   1:  PR[GP1:91,2] = PR[GP1:90,2] + -31.006;
   1:L PR[91] 10mm/sec CNT100;
   1:  PR[GP1:91,1] = PR[GP1:90,1] + -0.266;
   1:  PR[GP1:91,2] = PR[GP1:90,2] + -30.252;
   1:L PR[91] 10mm/sec CNT100;
   1:  PR[GP1:91,1] = PR[GP1:90,1] + 0.371;
   1:  PR[GP1:91,2] = PR[GP1:90,2] + -31.082;
   1:  PR[GP1:91,3] = PR[GP1:90,3] + 67.405;
   1:L PR[91] 10mm/sec CNT100;
   1:  PR[GP1:91,1] = PR[GP1:90,1] + 7.171;
   1:  PR[GP1:91,2] = PR[GP1:90,2] + -35.054;
   1:L PR[91] 10mm/sec CNT100;
   1:  PR[GP1:91,1] = PR[GP1:90,1] + 10.495;
   1:  PR[GP1:91,2] = PR[GP1:90,2] + -36.009;
   1:L PR[91] 10mm/sec CNT100;
   1:  PR[GP1:91,1] = PR[GP1:90,1] + 18.333;
   1:  PR[GP1:91,2] = PR[GP1:90,2] + -37.802;
   1:L PR[91] 10mm/sec CNT100;
   1:  PR[GP1:91,1] = PR[GP1:90,1] + 22.053;
   1:  PR[GP1:91,2] = PR[GP1:90,2] + -38.049;
   1:L PR[91] 10mm/sec CNT100;
   1:  PR[GP1:91,1] = PR[GP1:90,1] + 26.238;
   1:  PR[GP1:91,2] = PR[GP1:90,2] + -37.472;
   1:L PR[91] 10mm/sec CNT100;
   1:  PR[GP1:91,1] = PR[GP1:90,1] + 33.369;
   1:  PR[GP1:91,2] = PR[GP1:90,2] + -36.778;
   1:L PR[91] 10mm/sec CNT100;
   1:  PR[GP1:91,1] = PR[GP1:90,1] + 37.578;
   1:  PR[GP1:91,2] = PR[GP1:90,2] + -35.242;
   1:L PR[91] 10mm/sec CNT100;
   1:  PR[GP1:91,1] = PR[GP1:90,1] + 43.414;
   1:  PR[GP1:91,2] = PR[GP1:90,2] + -32.676;
   1:L PR[91] 10mm/sec CNT100;
   1:  PR[GP1:91,1] = PR[GP1:90,1] + 47.360;
   1:  PR[GP1:91,2] = PR[GP1:90,2] + -30.200;
   1:L PR[91] 10mm/sec CNT100;
   1:  PR[GP1:91,1] = PR[GP1:90,1] + 50.959;
   1:  PR[GP1:91,2] = PR[GP1:90,2] + -26.692;
   1:L PR[91] 10mm/sec CNT100;
   1:  PR[GP1:91,1] = PR[GP1:90,1] + 54.991;
   1:  PR[GP1:91,2] = PR[GP1:90,2] + -23.025;
   1:L PR[91] 10mm/sec CNT100;
   1:  PR[GP1:91,1] = PR[GP1:90,1] + 57.831;
   1:  PR[GP1:91,2] = PR[GP1:90,2] + -18.619;
   1:L PR[91] 10mm/sec CNT100;
   1:  PR[GP1:91,1] = PR[GP1:90,1] + 60.207;
   1:  PR[GP1:91,2] = PR[GP1:90,2] + -14.324;
   1:L PR[91] 10mm/sec CNT100;
   1:  PR[GP1:91,1] = PR[GP1:90,1] + 61.985;
   1:  PR[GP1:91,2] = PR[GP1:90,2] + -9.491;
   1:L PR[91] 10mm/sec CNT100;
   1:  PR[GP1:91,1] = PR[GP1:90,1] + 62.584;
   1:  PR[GP1:91,2] = PR[GP1:90,2] + -4.219;
   1:L PR[91] 10mm/sec CNT100;
   1:  PR[GP1:91,1] = PR[GP1:90,1] + 63.354;
   1:  PR[GP1:91,2] = PR[GP1:90,2] + 0.296;
   1:L PR[91] 10mm/sec CNT100;
   1:  PR[GP1:91,1] = PR[GP1:90,1] + 62.767;
   1:  PR[GP1:91,2] = PR[GP1:90,2] + 5.490;
   1:L PR[91] 10mm/sec CNT100;
   1:  PR[GP1:91,1] = PR[GP1:90,1] + 61.988;
   1:  PR[GP1:91,2] = PR[GP1:90,2] + 10.042;
   1:L PR[91] 10mm/sec CNT100;
   1:  PR[GP1:91,1] = PR[GP1:90,1] + 60.204;
   1:  PR[GP1:91,2] = PR[GP1:90,2] + 14.892;
   1:L PR[91] 10mm/sec CNT100;
   1:  PR[GP1:91,1] = PR[GP1:90,1] + 57.818;
   1:  PR[GP1:91,2] = PR[GP1:90,2] + 19.195;
   1:L PR[91] 10mm/sec CNT100;
   1:  PR[GP1:91,1] = PR[GP1:90,1] + 54.971;
   1:  PR[GP1:91,2] = PR[GP1:90,2] + 23.610;
   1:L PR[91] 10mm/sec CNT100;
   1:  PR[GP1:91,1] = PR[GP1:90,1] + 51.546;
   1:  PR[GP1:91,2] = PR[GP1:90,2] + 26.964;
   1:L PR[91] 10mm/sec CNT100;
   1:  PR[GP1:91,1] = PR[GP1:90,1] + 47.338;
   1:  PR[GP1:91,2] = PR[GP1:90,2] + 30.773;
   1:L PR[91] 10mm/sec CNT100;
   1:  PR[GP1:91,1] = PR[GP1:90,1] + 43.381;
   1:  PR[GP1:91,2] = PR[GP1:90,2] + 33.255;
   1:L PR[91] 10mm/sec CNT100;
   1:  PR[GP1:91,1] = PR[GP1:90,1] + 37.523;
   1:  PR[GP1:91,2] = PR[GP1:90,2] + 35.815;
   1:L PR[91] 10mm/sec CNT100;
   1:  PR[GP1:91,1] = PR[GP1:90,1] + 33.299;
   1:  PR[GP1:91,2] = PR[GP1:90,2] + 37.356;
   1:L PR[91] 10mm/sec CNT100;
   1:  PR[GP1:91,1] = PR[GP1:90,1] + 29.302;
   1:  PR[GP1:91,2] = PR[GP1:90,2] + 37.923;
   1:L PR[91] 10mm/sec CNT100;
   1:  PR[GP1:91,1] = PR[GP1:90,1] + 21.984;
   1:  PR[GP1:91,2] = PR[GP1:90,2] + 38.603;
   1:L PR[91] 10mm/sec CNT100;
   1:  PR[GP1:91,1] = PR[GP1:90,1] + 18.251;
   1:  PR[GP1:91,2] = PR[GP1:90,2] + 38.355;
   1:L PR[91] 10mm/sec CNT100;
   1:  PR[GP1:91,1] = PR[GP1:90,1] + 10.284;
   1:  PR[GP1:91,2] = PR[GP1:90,2] + 36.473;
   1:L PR[91] 10mm/sec CNT100;
   1:  PR[GP1:91,1] = PR[GP1:90,1] + 7.009;
   1:  PR[GP1:91,2] = PR[GP1:90,2] + 35.532;
   1:L PR[91] 10mm/sec CNT100;
   1:  PR[GP1:91,1] = PR[GP1:90,1] + 5.914;
   1:  PR[GP1:91,2] = PR[GP1:90,2] + 34.958;
   1:L PR[91] 10mm/sec CNT100;
   1:  PR[GP1:91,1] = PR[GP1:90,1] + 3.650;
   1:  PR[GP1:91,2] = PR[GP1:90,2] + 33.735;
   1:L PR[91] 10mm/sec CNT100;
   1:  PR[GP1:91,1] = PR[GP1:90,1] + -0.263;
   1:  PR[GP1:91,2] = PR[GP1:90,2] + 30.552;
   1:L PR[91] 10mm/sec CNT100;
   1:  PR[GP1:91,1] = PR[GP1:90,1] + -4.166;
   1:  PR[GP1:91,2] = PR[GP1:90,2] + 33.726;
   1:L PR[91] 10mm/sec CNT100;
   1:  PR[GP1:91,1] = PR[GP1:90,1] + -6.444;
   1:  PR[GP1:91,2] = PR[GP1:90,2] + 34.959;
   1:L PR[91] 10mm/sec CNT100;
   1:  PR[GP1:91,1] = PR[GP1:90,1] + -7.536;
   1:  PR[GP1:91,2] = PR[GP1:90,2] + 35.533;
   1:L PR[91] 10mm/sec CNT100;
   1:  PR[GP1:91,1] = PR[GP1:90,1] + -10.806;
   1:  PR[GP1:91,2] = PR[GP1:90,2] + 36.474;
   1:L PR[91] 10mm/sec CNT100;
   1:  PR[GP1:91,1] = PR[GP1:90,1] + -18.776;
   1:  PR[GP1:91,2] = PR[GP1:90,2] + 38.355;
   1:L PR[91] 10mm/sec CNT100;
   1:  PR[GP1:91,1] = PR[GP1:90,1] + -22.506;
   1:  PR[GP1:91,2] = PR[GP1:90,2] + 38.601;
   1:L PR[91] 10mm/sec CNT100;
   1:  PR[GP1:91,1] = PR[GP1:90,1] + -26.707;
   1:  PR[GP1:91,2] = PR[GP1:90,2] + 38.020;
   1:L PR[91] 10mm/sec CNT100;
   1:  PR[GP1:91,1] = PR[GP1:90,1] + -33.861;
   1:  PR[GP1:91,2] = PR[GP1:90,2] + 37.347;
   1:L PR[91] 10mm/sec CNT100;
   1:  PR[GP1:91,1] = PR[GP1:90,1] + -38.066;
   1:  PR[GP1:91,2] = PR[GP1:90,2] + 35.807;
   1:L PR[91] 10mm/sec CNT100;
   1:  PR[GP1:91,1] = PR[GP1:90,1] + -43.923;
   1:  PR[GP1:91,2] = PR[GP1:90,2] + 33.246;
   1:L PR[91] 10mm/sec CNT100;
   1:  PR[GP1:91,1] = PR[GP1:90,1] + -47.894;
   1:  PR[GP1:91,2] = PR[GP1:90,2] + 30.742;
   1:L PR[91] 10mm/sec CNT100;
   1:  PR[GP1:91,1] = PR[GP1:90,1] + -51.502;
   1:  PR[GP1:91,2] = PR[GP1:90,2] + 27.221;
   1:L PR[91] 10mm/sec CNT100;
   1:  PR[GP1:91,1] = PR[GP1:90,1] + -55.548;
   1:  PR[GP1:91,2] = PR[GP1:90,2] + 23.557;
   1:L PR[91] 10mm/sec CNT100;
   1:  PR[GP1:91,1] = PR[GP1:90,1] + -58.358;
   1:  PR[GP1:91,2] = PR[GP1:90,2] + 19.171;
   1:L PR[91] 10mm/sec CNT100;
   1:  PR[GP1:91,1] = PR[GP1:90,1] + -60.744;
   1:  PR[GP1:91,2] = PR[GP1:90,2] + 14.862;
   1:L PR[91] 10mm/sec CNT100;
   1:  PR[GP1:91,1] = PR[GP1:90,1] + -62.529;
   1:  PR[GP1:91,2] = PR[GP1:90,2] + 9.943;
   1:L PR[91] 10mm/sec CNT100;
   1:  PR[GP1:91,1] = PR[GP1:90,1] + -63.107;
   1:  PR[GP1:91,2] = PR[GP1:90,2] + 4.782;
   1:L PR[91] 10mm/sec CNT100;
   1:  PR[GP1:91,1] = PR[GP1:90,1] + -63.881;
   1:  PR[GP1:91,2] = PR[GP1:90,2] + 0.261;
   1:L PR[91] 10mm/sec CNT100;
   1:  PR[GP1:91,1] = PR[GP1:90,1] + -63.314;
   1:  PR[GP1:91,2] = PR[GP1:90,2] + -4.822;
   1:L PR[91] 10mm/sec CNT100;
   1:  PR[GP1:91,1] = PR[GP1:90,1] + -62.538;
   1:  PR[GP1:91,2] = PR[GP1:90,2] + -9.359;
   1:L PR[91] 10mm/sec CNT100;
   1:  PR[GP1:91,1] = PR[GP1:90,1] + -60.747;
   1:  PR[GP1:91,2] = PR[GP1:90,2] + -14.294;
   1:L PR[91] 10mm/sec CNT100;
   1:  PR[GP1:91,1] = PR[GP1:90,1] + -58.372;
   1:  PR[GP1:91,2] = PR[GP1:90,2] + -18.596;
   1:L PR[91] 10mm/sec CNT100;
   1:  PR[GP1:91,1] = PR[GP1:90,1] + -55.555;
   1:  PR[GP1:91,2] = PR[GP1:90,2] + -22.992;
   1:L PR[91] 10mm/sec CNT100;
   1:  PR[GP1:91,1] = PR[GP1:90,1] + -52.126;
   1:  PR[GP1:91,2] = PR[GP1:90,2] + -26.357;
   1:L PR[91] 10mm/sec CNT100;
   1:  PR[GP1:91,1] = PR[GP1:90,1] + -47.936;
   1:  PR[GP1:91,2] = PR[GP1:90,2] + -30.157;
   1:L PR[91] 10mm/sec CNT100;
   1:  PR[GP1:91,1] = PR[GP1:90,1] + -43.956;
   1:  PR[GP1:91,2] = PR[GP1:90,2] + -32.667;
   1:L PR[91] 10mm/sec CNT100;
   1:  PR[GP1:91,1] = PR[GP1:90,1] + -38.121;
   1:  PR[GP1:91,2] = PR[GP1:90,2] + -35.235;
   1:L PR[91] 10mm/sec CNT100;
   1:  PR[GP1:91,1] = PR[GP1:90,1] + -33.905;
   1:  PR[GP1:91,2] = PR[GP1:90,2] + -36.779;
   1:L PR[91] 10mm/sec CNT100;
   1:  PR[GP1:91,1] = PR[GP1:90,1] + -29.897;
   1:  PR[GP1:91,2] = PR[GP1:90,2] + -37.349;
   1:L PR[91] 10mm/sec CNT100;
   1:  PR[GP1:91,1] = PR[GP1:90,1] + -22.602;
   1:  PR[GP1:91,2] = PR[GP1:90,2] + -38.049;
   1:L PR[91] 10mm/sec CNT100;
   1:  PR[GP1:91,1] = PR[GP1:90,1] + -18.858;
   1:  PR[GP1:91,2] = PR[GP1:90,2] + -37.802;
   1:L PR[91] 10mm/sec CNT100;
   1:  PR[GP1:91,1] = PR[GP1:90,1] + -11.020;
   1:  PR[GP1:91,2] = PR[GP1:90,2] + -36.009;
   1:L PR[91] 10mm/sec CNT100;
   1:  PR[GP1:91,1] = PR[GP1:90,1] + -7.700;
   1:  PR[GP1:91,2] = PR[GP1:90,2] + -35.055;
   1:L PR[91] 10mm/sec CNT100;
   1:  PR[GP1:91,1] = PR[GP1:90,1] + -0.903;
   1:  PR[GP1:91,2] = PR[GP1:90,2] + -31.081;
   1:L PR[91] 10mm/sec CNT100;
   1:  PR[GP1:91,1] = PR[GP1:90,1] + -0.266;
   1:  PR[GP1:91,2] = PR[GP1:90,2] + -30.532;
   1:L PR[91] 10mm/sec CNT100;
   1:  PR[GP1:91,1] = PR[GP1:90,1] + 0.126;
   1:  PR[GP1:91,2] = PR[GP1:90,2] + -31.151;
   1:  PR[GP1:91,3] = PR[GP1:90,3] + 68.015;
   1:L PR[91] 10mm/sec CNT100;
   1:  PR[GP1:91,1] = PR[GP1:90,1] + 6.916;
   1:  PR[GP1:91,2] = PR[GP1:90,2] + -35.123;
   1:L PR[91] 10mm/sec CNT100;
   1:  PR[GP1:91,1] = PR[GP1:90,1] + 10.120;
   1:  PR[GP1:91,2] = PR[GP1:90,2] + -36.043;
   1:L PR[91] 10mm/sec CNT100;
   1:  PR[GP1:91,1] = PR[GP1:90,1] + 18.156;
   1:  PR[GP1:91,2] = PR[GP1:90,2] + -37.882;
   1:L PR[91] 10mm/sec CNT100;
   1:  PR[GP1:91,1] = PR[GP1:90,1] + 21.753;
   1:  PR[GP1:91,2] = PR[GP1:90,2] + -38.121;
   1:L PR[91] 10mm/sec CNT100;
   1:  PR[GP1:91,1] = PR[GP1:90,1] + 25.802;
   1:  PR[GP1:91,2] = PR[GP1:90,2] + -37.562;
   1:L PR[91] 10mm/sec CNT100;
   1:  PR[GP1:91,1] = PR[GP1:90,1] + 33.152;
   1:  PR[GP1:91,2] = PR[GP1:90,2] + -36.848;
   1:L PR[91] 10mm/sec CNT100;
   1:  PR[GP1:91,1] = PR[GP1:90,1] + 37.234;
   1:  PR[GP1:91,2] = PR[GP1:90,2] + -35.358;
   1:L PR[91] 10mm/sec CNT100;
   1:  PR[GP1:91,1] = PR[GP1:90,1] + 43.269;
   1:  PR[GP1:91,2] = PR[GP1:90,2] + -32.704;
   1:L PR[91] 10mm/sec CNT100;
   1:  PR[GP1:91,1] = PR[GP1:90,1] + 47.105;
   1:  PR[GP1:91,2] = PR[GP1:90,2] + -30.297;
   1:L PR[91] 10mm/sec CNT100;
   1:  PR[GP1:91,1] = PR[GP1:90,1] + 50.604;
   1:  PR[GP1:91,2] = PR[GP1:90,2] + -26.887;
   1:L PR[91] 10mm/sec CNT100;
   1:  PR[GP1:91,1] = PR[GP1:90,1] + 54.804;
   1:  PR[GP1:91,2] = PR[GP1:90,2] + -23.066;
   1:L PR[91] 10mm/sec CNT100;
   1:  PR[GP1:91,1] = PR[GP1:90,1] + 57.569;
   1:  PR[GP1:91,2] = PR[GP1:90,2] + -18.777;
   1:L PR[91] 10mm/sec CNT100;
   1:  PR[GP1:91,1] = PR[GP1:90,1] + 60.053;
   1:  PR[GP1:91,2] = PR[GP1:90,2] + -14.287;
   1:L PR[91] 10mm/sec CNT100;
   1:  PR[GP1:91,1] = PR[GP1:90,1] + 61.786;
   1:  PR[GP1:91,2] = PR[GP1:90,2] + -9.578;
   1:L PR[91] 10mm/sec CNT100;
   1:  PR[GP1:91,1] = PR[GP1:90,1] + 62.370;
   1:  PR[GP1:91,2] = PR[GP1:90,2] + -4.439;
   1:L PR[91] 10mm/sec CNT100;
   1:  PR[GP1:91,1] = PR[GP1:90,1] + 63.177;
   1:  PR[GP1:91,2] = PR[GP1:90,2] + 0.296;
   1:L PR[91] 10mm/sec CNT100;
   1:  PR[GP1:91,1] = PR[GP1:90,1] + 62.605;
   1:  PR[GP1:91,2] = PR[GP1:90,2] + 5.360;
   1:L PR[91] 10mm/sec CNT100;
   1:  PR[GP1:91,1] = PR[GP1:90,1] + 61.788;
   1:  PR[GP1:91,2] = PR[GP1:90,2] + 10.130;
   1:L PR[91] 10mm/sec CNT100;
   1:  PR[GP1:91,1] = PR[GP1:90,1] + 60.050;
   1:  PR[GP1:91,2] = PR[GP1:90,2] + 14.855;
   1:L PR[91] 10mm/sec CNT100;
   1:  PR[GP1:91,1] = PR[GP1:90,1] + 57.555;
   1:  PR[GP1:91,2] = PR[GP1:90,2] + 19.353;
   1:L PR[91] 10mm/sec CNT100;
   1:  PR[GP1:91,1] = PR[GP1:90,1] + 54.783;
   1:  PR[GP1:91,2] = PR[GP1:90,2] + 23.653;
   1:L PR[91] 10mm/sec CNT100;
   1:  PR[GP1:91,1] = PR[GP1:90,1] + 51.448;
   1:  PR[GP1:91,2] = PR[GP1:90,2] + 26.918;
   1:L PR[91] 10mm/sec CNT100;
   1:  PR[GP1:91,1] = PR[GP1:90,1] + 47.081;
   1:  PR[GP1:91,2] = PR[GP1:90,2] + 30.871;
   1:L PR[91] 10mm/sec CNT100;
   1:  PR[GP1:91,1] = PR[GP1:90,1] + 43.235;
   1:  PR[GP1:91,2] = PR[GP1:90,2] + 33.284;
   1:L PR[91] 10mm/sec CNT100;
   1:  PR[GP1:91,1] = PR[GP1:90,1] + 37.177;
   1:  PR[GP1:91,2] = PR[GP1:90,2] + 35.931;
   1:L PR[91] 10mm/sec CNT100;
   1:  PR[GP1:91,1] = PR[GP1:90,1] + 33.080;
   1:  PR[GP1:91,2] = PR[GP1:90,2] + 37.426;
   1:L PR[91] 10mm/sec CNT100;
   1:  PR[GP1:91,1] = PR[GP1:90,1] + 29.203;
   1:  PR[GP1:91,2] = PR[GP1:90,2] + 37.976;
   1:L PR[91] 10mm/sec CNT100;
   1:  PR[GP1:91,1] = PR[GP1:90,1] + 21.682;
   1:  PR[GP1:91,2] = PR[GP1:90,2] + 38.675;
   1:L PR[91] 10mm/sec CNT100;
   1:  PR[GP1:91,1] = PR[GP1:90,1] + 18.072;
   1:  PR[GP1:91,2] = PR[GP1:90,2] + 38.435;
   1:L PR[91] 10mm/sec CNT100;
   1:  PR[GP1:91,1] = PR[GP1:90,1] + 9.904;
   1:  PR[GP1:91,2] = PR[GP1:90,2] + 36.506;
   1:L PR[91] 10mm/sec CNT100;
   1:  PR[GP1:91,1] = PR[GP1:90,1] + 6.751;
   1:  PR[GP1:91,2] = PR[GP1:90,2] + 35.599;
   1:L PR[91] 10mm/sec CNT100;
   1:  PR[GP1:91,1] = PR[GP1:90,1] + 5.630;
   1:  PR[GP1:91,2] = PR[GP1:90,2] + 35.011;
   1:L PR[91] 10mm/sec CNT100;
   1:  PR[GP1:91,1] = PR[GP1:90,1] + 3.477;
   1:  PR[GP1:91,2] = PR[GP1:90,2] + 33.849;
   1:L PR[91] 10mm/sec CNT100;
   1:  PR[GP1:91,1] = PR[GP1:90,1] + -0.263;
   1:  PR[GP1:91,2] = PR[GP1:90,2] + 30.807;
   1:L PR[91] 10mm/sec CNT100;
   1:  PR[GP1:91,1] = PR[GP1:90,1] + -3.994;
   1:  PR[GP1:91,2] = PR[GP1:90,2] + 33.840;
   1:L PR[91] 10mm/sec CNT100;
   1:  PR[GP1:91,1] = PR[GP1:90,1] + -6.158;
   1:  PR[GP1:91,2] = PR[GP1:90,2] + 35.012;
   1:L PR[91] 10mm/sec CNT100;
   1:  PR[GP1:91,1] = PR[GP1:90,1] + -7.277;
   1:  PR[GP1:91,2] = PR[GP1:90,2] + 35.601;
   1:L PR[91] 10mm/sec CNT100;
   1:  PR[GP1:91,1] = PR[GP1:90,1] + -10.426;
   1:  PR[GP1:91,2] = PR[GP1:90,2] + 36.506;
   1:L PR[91] 10mm/sec CNT100;
   1:  PR[GP1:91,1] = PR[GP1:90,1] + -18.597;
   1:  PR[GP1:91,2] = PR[GP1:90,2] + 38.435;
   1:L PR[91] 10mm/sec CNT100;
   1:  PR[GP1:91,1] = PR[GP1:90,1] + -22.204;
   1:  PR[GP1:91,2] = PR[GP1:90,2] + 38.673;
   1:L PR[91] 10mm/sec CNT100;
   1:  PR[GP1:91,1] = PR[GP1:90,1] + -26.268;
   1:  PR[GP1:91,2] = PR[GP1:90,2] + 38.111;
   1:L PR[91] 10mm/sec CNT100;
   1:  PR[GP1:91,1] = PR[GP1:90,1] + -33.641;
   1:  PR[GP1:91,2] = PR[GP1:90,2] + 37.417;
   1:L PR[91] 10mm/sec CNT100;
   1:  PR[GP1:91,1] = PR[GP1:90,1] + -37.719;
   1:  PR[GP1:91,2] = PR[GP1:90,2] + 35.924;
   1:L PR[91] 10mm/sec CNT100;
   1:  PR[GP1:91,1] = PR[GP1:90,1] + -43.777;
   1:  PR[GP1:91,2] = PR[GP1:90,2] + 33.275;
   1:L PR[91] 10mm/sec CNT100;
   1:  PR[GP1:91,1] = PR[GP1:90,1] + -47.636;
   1:  PR[GP1:91,2] = PR[GP1:90,2] + 30.842;
   1:L PR[91] 10mm/sec CNT100;
   1:  PR[GP1:91,1] = PR[GP1:90,1] + -51.144;
   1:  PR[GP1:91,2] = PR[GP1:90,2] + 27.417;
   1:L PR[91] 10mm/sec CNT100;
   1:  PR[GP1:91,1] = PR[GP1:90,1] + -55.359;
   1:  PR[GP1:91,2] = PR[GP1:90,2] + 23.601;
   1:L PR[91] 10mm/sec CNT100;
   1:  PR[GP1:91,1] = PR[GP1:90,1] + -58.095;
   1:  PR[GP1:91,2] = PR[GP1:90,2] + 19.331;
   1:L PR[91] 10mm/sec CNT100;
   1:  PR[GP1:91,1] = PR[GP1:90,1] + -60.589;
   1:  PR[GP1:91,2] = PR[GP1:90,2] + 14.826;
   1:L PR[91] 10mm/sec CNT100;
   1:  PR[GP1:91,1] = PR[GP1:90,1] + -62.329;
   1:  PR[GP1:91,2] = PR[GP1:90,2] + 10.033;
   1:L PR[91] 10mm/sec CNT100;
   1:  PR[GP1:91,1] = PR[GP1:90,1] + -62.892;
   1:  PR[GP1:91,2] = PR[GP1:90,2] + 5.002;
   1:L PR[91] 10mm/sec CNT100;
   1:  PR[GP1:91,1] = PR[GP1:90,1] + -63.704;
   1:  PR[GP1:91,2] = PR[GP1:90,2] + 0.261;
   1:L PR[91] 10mm/sec CNT100;
   1:  PR[GP1:91,1] = PR[GP1:90,1] + -63.151;
   1:  PR[GP1:91,2] = PR[GP1:90,2] + -4.694;
   1:L PR[91] 10mm/sec CNT100;
   1:  PR[GP1:91,1] = PR[GP1:90,1] + -62.338;
   1:  PR[GP1:91,2] = PR[GP1:90,2] + -9.448;
   1:L PR[91] 10mm/sec CNT100;
   1:  PR[GP1:91,1] = PR[GP1:90,1] + -60.593;
   1:  PR[GP1:91,2] = PR[GP1:90,2] + -14.258;
   1:L PR[91] 10mm/sec CNT100;
   1:  PR[GP1:91,1] = PR[GP1:90,1] + -58.109;
   1:  PR[GP1:91,2] = PR[GP1:90,2] + -18.754;
   1:L PR[91] 10mm/sec CNT100;
   1:  PR[GP1:91,1] = PR[GP1:90,1] + -55.367;
   1:  PR[GP1:91,2] = PR[GP1:90,2] + -23.035;
   1:L PR[91] 10mm/sec CNT100;
   1:  PR[GP1:91,1] = PR[GP1:90,1] + -52.028;
   1:  PR[GP1:91,2] = PR[GP1:90,2] + -26.311;
   1:L PR[91] 10mm/sec CNT100;
   1:  PR[GP1:91,1] = PR[GP1:90,1] + -47.680;
   1:  PR[GP1:91,2] = PR[GP1:90,2] + -30.256;
   1:L PR[91] 10mm/sec CNT100;
   1:  PR[GP1:91,1] = PR[GP1:90,1] + -43.811;
   1:  PR[GP1:91,2] = PR[GP1:90,2] + -32.695;
   1:L PR[91] 10mm/sec CNT100;
   1:  PR[GP1:91,1] = PR[GP1:90,1] + -37.777;
   1:  PR[GP1:91,2] = PR[GP1:90,2] + -35.351;
   1:L PR[91] 10mm/sec CNT100;
   1:  PR[GP1:91,1] = PR[GP1:90,1] + -33.687;
   1:  PR[GP1:91,2] = PR[GP1:90,2] + -36.849;
   1:L PR[91] 10mm/sec CNT100;
   1:  PR[GP1:91,1] = PR[GP1:90,1] + -29.799;
   1:  PR[GP1:91,2] = PR[GP1:90,2] + -37.402;
   1:L PR[91] 10mm/sec CNT100;
   1:  PR[GP1:91,1] = PR[GP1:90,1] + -22.302;
   1:  PR[GP1:91,2] = PR[GP1:90,2] + -38.121;
   1:L PR[91] 10mm/sec CNT100;
   1:  PR[GP1:91,1] = PR[GP1:90,1] + -18.681;
   1:  PR[GP1:91,2] = PR[GP1:90,2] + -37.882;
   1:L PR[91] 10mm/sec CNT100;
   1:  PR[GP1:91,1] = PR[GP1:90,1] + -10.645;
   1:  PR[GP1:91,2] = PR[GP1:90,2] + -36.044;
   1:L PR[91] 10mm/sec CNT100;
   1:  PR[GP1:91,1] = PR[GP1:90,1] + -7.446;
   1:  PR[GP1:91,2] = PR[GP1:90,2] + -35.125;
   1:L PR[91] 10mm/sec CNT100;
   1:  PR[GP1:91,1] = PR[GP1:90,1] + -0.659;
   1:  PR[GP1:91,2] = PR[GP1:90,2] + -31.150;
   1:L PR[91] 10mm/sec CNT100;
   1:  PR[GP1:91,1] = PR[GP1:90,1] + -0.266;
   1:  PR[GP1:91,2] = PR[GP1:90,2] + -30.811;
   1:L PR[91] 10mm/sec CNT100;
   1:  PR[GP1:91,1] = PR[GP1:90,1] + 6.662;
   1:  PR[GP1:91,2] = PR[GP1:90,2] + -35.193;
   1:  PR[GP1:91,3] = PR[GP1:90,3] + 68.625;
   1:L PR[91] 10mm/sec CNT100;
   1:  PR[GP1:91,1] = PR[GP1:90,1] + 9.744;
   1:  PR[GP1:91,2] = PR[GP1:90,2] + -36.078;
   1:L PR[91] 10mm/sec CNT100;
   1:  PR[GP1:91,1] = PR[GP1:90,1] + 17.979;
   1:  PR[GP1:91,2] = PR[GP1:90,2] + -37.962;
   1:L PR[91] 10mm/sec CNT100;
   1:  PR[GP1:91,1] = PR[GP1:90,1] + 21.453;
   1:  PR[GP1:91,2] = PR[GP1:90,2] + -38.193;
   1:L PR[91] 10mm/sec CNT100;
   1:  PR[GP1:91,1] = PR[GP1:90,1] + 25.366;
   1:  PR[GP1:91,2] = PR[GP1:90,2] + -37.653;
   1:L PR[91] 10mm/sec CNT100;
   1:  PR[GP1:91,1] = PR[GP1:90,1] + 32.934;
   1:  PR[GP1:91,2] = PR[GP1:90,2] + -36.918;
   1:L PR[91] 10mm/sec CNT100;
   1:  PR[GP1:91,1] = PR[GP1:90,1] + 36.890;
   1:  PR[GP1:91,2] = PR[GP1:90,2] + -35.474;
   1:L PR[91] 10mm/sec CNT100;
   1:  PR[GP1:91,1] = PR[GP1:90,1] + 43.124;
   1:  PR[GP1:91,2] = PR[GP1:90,2] + -32.732;
   1:L PR[91] 10mm/sec CNT100;
   1:  PR[GP1:91,1] = PR[GP1:90,1] + 46.849;
   1:  PR[GP1:91,2] = PR[GP1:90,2] + -30.395;
   1:L PR[91] 10mm/sec CNT100;
   1:  PR[GP1:91,1] = PR[GP1:90,1] + 50.249;
   1:  PR[GP1:91,2] = PR[GP1:90,2] + -27.081;
   1:L PR[91] 10mm/sec CNT100;
   1:  PR[GP1:91,1] = PR[GP1:90,1] + 54.617;
   1:  PR[GP1:91,2] = PR[GP1:90,2] + -23.108;
   1:L PR[91] 10mm/sec CNT100;
   1:  PR[GP1:91,1] = PR[GP1:90,1] + 57.308;
   1:  PR[GP1:91,2] = PR[GP1:90,2] + -18.935;
   1:L PR[91] 10mm/sec CNT100;
   1:  PR[GP1:91,1] = PR[GP1:90,1] + 59.899;
   1:  PR[GP1:91,2] = PR[GP1:90,2] + -14.251;
   1:L PR[91] 10mm/sec CNT100;
   1:  PR[GP1:91,1] = PR[GP1:90,1] + 61.586;
   1:  PR[GP1:91,2] = PR[GP1:90,2] + -9.664;
   1:L PR[91] 10mm/sec CNT100;
   1:  PR[GP1:91,1] = PR[GP1:90,1] + 62.155;
   1:  PR[GP1:91,2] = PR[GP1:90,2] + -4.659;
   1:L PR[91] 10mm/sec CNT100;
   1:  PR[GP1:91,1] = PR[GP1:90,1] + 63.000;
   1:  PR[GP1:91,2] = PR[GP1:90,2] + 0.296;
   1:L PR[91] 10mm/sec CNT100;
   1:  PR[GP1:91,1] = PR[GP1:90,1] + 62.442;
   1:  PR[GP1:91,2] = PR[GP1:90,2] + 5.229;
   1:L PR[91] 10mm/sec CNT100;
   1:  PR[GP1:91,1] = PR[GP1:90,1] + 61.588;
   1:  PR[GP1:91,2] = PR[GP1:90,2] + 10.217;
   1:L PR[91] 10mm/sec CNT100;
   1:  PR[GP1:91,1] = PR[GP1:90,1] + 59.895;
   1:  PR[GP1:91,2] = PR[GP1:90,2] + 14.819;
   1:L PR[91] 10mm/sec CNT100;
   1:  PR[GP1:91,1] = PR[GP1:90,1] + 57.293;
   1:  PR[GP1:91,2] = PR[GP1:90,2] + 19.511;
   1:L PR[91] 10mm/sec CNT100;
   1:  PR[GP1:91,1] = PR[GP1:90,1] + 54.596;
   1:  PR[GP1:91,2] = PR[GP1:90,2] + 23.695;
   1:L PR[91] 10mm/sec CNT100;
   1:  PR[GP1:91,1] = PR[GP1:90,1] + 51.351;
   1:  PR[GP1:91,2] = PR[GP1:90,2] + 26.872;
   1:L PR[91] 10mm/sec CNT100;
   1:  PR[GP1:91,1] = PR[GP1:90,1] + 46.824;
   1:  PR[GP1:91,2] = PR[GP1:90,2] + 30.970;
   1:L PR[91] 10mm/sec CNT100;
   1:  PR[GP1:91,1] = PR[GP1:90,1] + 43.088;
   1:  PR[GP1:91,2] = PR[GP1:90,2] + 33.313;
   1:L PR[91] 10mm/sec CNT100;
   1:  PR[GP1:91,1] = PR[GP1:90,1] + 36.831;
   1:  PR[GP1:91,2] = PR[GP1:90,2] + 36.047;
   1:L PR[91] 10mm/sec CNT100;
   1:  PR[GP1:91,1] = PR[GP1:90,1] + 32.861;
   1:  PR[GP1:91,2] = PR[GP1:90,2] + 37.496;
   1:L PR[91] 10mm/sec CNT100;
   1:  PR[GP1:91,1] = PR[GP1:90,1] + 29.104;
   1:  PR[GP1:91,2] = PR[GP1:90,2] + 38.029;
   1:L PR[91] 10mm/sec CNT100;
   1:  PR[GP1:91,1] = PR[GP1:90,1] + 21.379;
   1:  PR[GP1:91,2] = PR[GP1:90,2] + 38.747;
   1:L PR[91] 10mm/sec CNT100;
   1:  PR[GP1:91,1] = PR[GP1:90,1] + 17.893;
   1:  PR[GP1:91,2] = PR[GP1:90,2] + 38.515;
   1:L PR[91] 10mm/sec CNT100;
   1:  PR[GP1:91,1] = PR[GP1:90,1] + 9.523;
   1:  PR[GP1:91,2] = PR[GP1:90,2] + 36.538;
   1:L PR[91] 10mm/sec CNT100;
   1:  PR[GP1:91,1] = PR[GP1:90,1] + 6.493;
   1:  PR[GP1:91,2] = PR[GP1:90,2] + 35.667;
   1:L PR[91] 10mm/sec CNT100;
   1:  PR[GP1:91,1] = PR[GP1:90,1] + 5.344;
   1:  PR[GP1:91,2] = PR[GP1:90,2] + 35.065;
   1:L PR[91] 10mm/sec CNT100;
   1:  PR[GP1:91,1] = PR[GP1:90,1] + 3.304;
   1:  PR[GP1:91,2] = PR[GP1:90,2] + 33.963;
   1:L PR[91] 10mm/sec CNT100;
   1:  PR[GP1:91,1] = PR[GP1:90,1] + -0.263;
   1:  PR[GP1:91,2] = PR[GP1:90,2] + 31.062;
   1:L PR[91] 10mm/sec CNT100;
   1:  PR[GP1:91,1] = PR[GP1:90,1] + -3.821;
   1:  PR[GP1:91,2] = PR[GP1:90,2] + 33.955;
   1:L PR[91] 10mm/sec CNT100;
   1:  PR[GP1:91,1] = PR[GP1:90,1] + -5.873;
   1:  PR[GP1:91,2] = PR[GP1:90,2] + 35.066;
   1:L PR[91] 10mm/sec CNT100;
   1:  PR[GP1:91,1] = PR[GP1:90,1] + -7.019;
   1:  PR[GP1:91,2] = PR[GP1:90,2] + 35.668;
   1:L PR[91] 10mm/sec CNT100;
   1:  PR[GP1:91,1] = PR[GP1:90,1] + -10.045;
   1:  PR[GP1:91,2] = PR[GP1:90,2] + 36.538;
   1:L PR[91] 10mm/sec CNT100;
   1:  PR[GP1:91,1] = PR[GP1:90,1] + -18.418;
   1:  PR[GP1:91,2] = PR[GP1:90,2] + 38.515;
   1:L PR[91] 10mm/sec CNT100;
   1:  PR[GP1:91,1] = PR[GP1:90,1] + -21.901;
   1:  PR[GP1:91,2] = PR[GP1:90,2] + 38.745;
   1:L PR[91] 10mm/sec CNT100;
   1:  PR[GP1:91,1] = PR[GP1:90,1] + -25.829;
   1:  PR[GP1:91,2] = PR[GP1:90,2] + 38.201;
   1:L PR[91] 10mm/sec CNT100;
   1:  PR[GP1:91,1] = PR[GP1:90,1] + -33.421;
   1:  PR[GP1:91,2] = PR[GP1:90,2] + 37.488;
   1:L PR[91] 10mm/sec CNT100;
   1:  PR[GP1:91,1] = PR[GP1:90,1] + -37.373;
   1:  PR[GP1:91,2] = PR[GP1:90,2] + 36.040;
   1:L PR[91] 10mm/sec CNT100;
   1:  PR[GP1:91,1] = PR[GP1:90,1] + -43.630;
   1:  PR[GP1:91,2] = PR[GP1:90,2] + 33.305;
   1:L PR[91] 10mm/sec CNT100;
   1:  PR[GP1:91,1] = PR[GP1:90,1] + -47.379;
   1:  PR[GP1:91,2] = PR[GP1:90,2] + 30.941;
   1:L PR[91] 10mm/sec CNT100;
   1:  PR[GP1:91,1] = PR[GP1:90,1] + -50.786;
   1:  PR[GP1:91,2] = PR[GP1:90,2] + 27.614;
   1:L PR[91] 10mm/sec CNT100;
   1:  PR[GP1:91,1] = PR[GP1:90,1] + -55.170;
   1:  PR[GP1:91,2] = PR[GP1:90,2] + 23.645;
   1:L PR[91] 10mm/sec CNT100;
   1:  PR[GP1:91,1] = PR[GP1:90,1] + -57.832;
   1:  PR[GP1:91,2] = PR[GP1:90,2] + 19.490;
   1:L PR[91] 10mm/sec CNT100;
   1:  PR[GP1:91,1] = PR[GP1:90,1] + -60.434;
   1:  PR[GP1:91,2] = PR[GP1:90,2] + 14.790;
   1:L PR[91] 10mm/sec CNT100;
   1:  PR[GP1:91,1] = PR[GP1:90,1] + -62.129;
   1:  PR[GP1:91,2] = PR[GP1:90,2] + 10.122;
   1:L PR[91] 10mm/sec CNT100;
   1:  PR[GP1:91,1] = PR[GP1:90,1] + -62.677;
   1:  PR[GP1:91,2] = PR[GP1:90,2] + 5.222;
   1:L PR[91] 10mm/sec CNT100;
   1:  PR[GP1:91,1] = PR[GP1:90,1] + -63.526;
   1:  PR[GP1:91,2] = PR[GP1:90,2] + 0.261;
   1:L PR[91] 10mm/sec CNT100;
   1:  PR[GP1:91,1] = PR[GP1:90,1] + -62.989;
   1:  PR[GP1:91,2] = PR[GP1:90,2] + -4.566;
   1:L PR[91] 10mm/sec CNT100;
   1:  PR[GP1:91,1] = PR[GP1:90,1] + -62.138;
   1:  PR[GP1:91,2] = PR[GP1:90,2] + -9.537;
   1:L PR[91] 10mm/sec CNT100;
   1:  PR[GP1:91,1] = PR[GP1:90,1] + -60.438;
   1:  PR[GP1:91,2] = PR[GP1:90,2] + -14.221;
   1:L PR[91] 10mm/sec CNT100;
   1:  PR[GP1:91,1] = PR[GP1:90,1] + -57.847;
   1:  PR[GP1:91,2] = PR[GP1:90,2] + -18.913;
   1:L PR[91] 10mm/sec CNT100;
   1:  PR[GP1:91,1] = PR[GP1:90,1] + -55.179;
   1:  PR[GP1:91,2] = PR[GP1:90,2] + -23.077;
   1:L PR[91] 10mm/sec CNT100;
   1:  PR[GP1:91,1] = PR[GP1:90,1] + -51.930;
   1:  PR[GP1:91,2] = PR[GP1:90,2] + -26.265;
   1:L PR[91] 10mm/sec CNT100;
   1:  PR[GP1:91,1] = PR[GP1:90,1] + -47.423;
   1:  PR[GP1:91,2] = PR[GP1:90,2] + -30.354;
   1:L PR[91] 10mm/sec CNT100;
   1:  PR[GP1:91,1] = PR[GP1:90,1] + -43.665;
   1:  PR[GP1:91,2] = PR[GP1:90,2] + -32.724;
   1:L PR[91] 10mm/sec CNT100;
   1:  PR[GP1:91,1] = PR[GP1:90,1] + -37.432;
   1:  PR[GP1:91,2] = PR[GP1:90,2] + -35.467;
   1:L PR[91] 10mm/sec CNT100;
   1:  PR[GP1:91,1] = PR[GP1:90,1] + -33.469;
   1:  PR[GP1:91,2] = PR[GP1:90,2] + -36.918;
   1:L PR[91] 10mm/sec CNT100;
   1:  PR[GP1:91,1] = PR[GP1:90,1] + -29.701;
   1:  PR[GP1:91,2] = PR[GP1:90,2] + -37.455;
   1:L PR[91] 10mm/sec CNT100;
   1:  PR[GP1:91,1] = PR[GP1:90,1] + -22.002;
   1:  PR[GP1:91,2] = PR[GP1:90,2] + -38.193;
   1:L PR[91] 10mm/sec CNT100;
   1:  PR[GP1:91,1] = PR[GP1:90,1] + -18.504;
   1:  PR[GP1:91,2] = PR[GP1:90,2] + -37.962;
   1:L PR[91] 10mm/sec CNT100;
   1:  PR[GP1:91,1] = PR[GP1:90,1] + -10.269;
   1:  PR[GP1:91,2] = PR[GP1:90,2] + -36.078;
   1:L PR[91] 10mm/sec CNT100;
   1:  PR[GP1:91,1] = PR[GP1:90,1] + -7.191;
   1:  PR[GP1:91,2] = PR[GP1:90,2] + -35.194;
   1:L PR[91] 10mm/sec CNT100;
   1:  PR[GP1:91,1] = PR[GP1:90,1] + -0.267;
   1:  PR[GP1:91,2] = PR[GP1:90,2] + -31.138;
   1:L PR[91] 10mm/sec CNT100;
   1:  PR[GP1:91,1] = PR[GP1:90,1] + 6.407;
   1:  PR[GP1:91,2] = PR[GP1:90,2] + -35.262;
   1:  PR[GP1:91,3] = PR[GP1:90,3] + 69.235;
   1:L PR[91] 10mm/sec CNT100;
   1:  PR[GP1:91,1] = PR[GP1:90,1] + 9.369;
   1:  PR[GP1:91,2] = PR[GP1:90,2] + -36.113;
   1:L PR[91] 10mm/sec CNT100;
   1:  PR[GP1:91,1] = PR[GP1:90,1] + 17.803;
   1:  PR[GP1:91,2] = PR[GP1:90,2] + -38.043;
   1:L PR[91] 10mm/sec CNT100;
   1:  PR[GP1:91,1] = PR[GP1:90,1] + 21.153;
   1:  PR[GP1:91,2] = PR[GP1:90,2] + -38.265;
   1:L PR[91] 10mm/sec CNT100;
   1:  PR[GP1:91,1] = PR[GP1:90,1] + 24.930;
   1:  PR[GP1:91,2] = PR[GP1:90,2] + -37.744;
   1:L PR[91] 10mm/sec CNT100;
   1:  PR[GP1:91,1] = PR[GP1:90,1] + 32.717;
   1:  PR[GP1:91,2] = PR[GP1:90,2] + -36.987;
   1:L PR[91] 10mm/sec CNT100;
   1:  PR[GP1:91,1] = PR[GP1:90,1] + 36.546;
   1:  PR[GP1:91,2] = PR[GP1:90,2] + -35.590;
   1:L PR[91] 10mm/sec CNT100;
   1:  PR[GP1:91,1] = PR[GP1:90,1] + 42.978;
   1:  PR[GP1:91,2] = PR[GP1:90,2] + -32.761;
   1:L PR[91] 10mm/sec CNT100;
   1:  PR[GP1:91,1] = PR[GP1:90,1] + 46.594;
   1:  PR[GP1:91,2] = PR[GP1:90,2] + -30.493;
   1:L PR[91] 10mm/sec CNT100;
   1:  PR[GP1:91,1] = PR[GP1:90,1] + 49.894;
   1:  PR[GP1:91,2] = PR[GP1:90,2] + -27.276;
   1:L PR[91] 10mm/sec CNT100;
   1:  PR[GP1:91,1] = PR[GP1:90,1] + 54.430;
   1:  PR[GP1:91,2] = PR[GP1:90,2] + -23.150;
   1:L PR[91] 10mm/sec CNT100;
   1:  PR[GP1:91,1] = PR[GP1:90,1] + 57.046;
   1:  PR[GP1:91,2] = PR[GP1:90,2] + -19.092;
   1:L PR[91] 10mm/sec CNT100;
   1:  PR[GP1:91,1] = PR[GP1:90,1] + 59.745;
   1:  PR[GP1:91,2] = PR[GP1:90,2] + -14.214;
   1:L PR[91] 10mm/sec CNT100;
   1:  PR[GP1:91,1] = PR[GP1:90,1] + 61.386;
   1:  PR[GP1:91,2] = PR[GP1:90,2] + -9.751;
   1:L PR[91] 10mm/sec CNT100;
   1:  PR[GP1:91,1] = PR[GP1:90,1] + 61.940;
   1:  PR[GP1:91,2] = PR[GP1:90,2] + -4.879;
   1:L PR[91] 10mm/sec CNT100;
   1:  PR[GP1:91,1] = PR[GP1:90,1] + 62.823;
   1:  PR[GP1:91,2] = PR[GP1:90,2] + 0.296;
   1:L PR[91] 10mm/sec CNT100;
   1:  PR[GP1:91,1] = PR[GP1:90,1] + 62.280;
   1:  PR[GP1:91,2] = PR[GP1:90,2] + 5.098;
   1:L PR[91] 10mm/sec CNT100;
   1:  PR[GP1:91,1] = PR[GP1:90,1] + 61.388;
   1:  PR[GP1:91,2] = PR[GP1:90,2] + 10.304;
   1:L PR[91] 10mm/sec CNT100;
   1:  PR[GP1:91,1] = PR[GP1:90,1] + 59.741;
   1:  PR[GP1:91,2] = PR[GP1:90,2] + 14.783;
   1:L PR[91] 10mm/sec CNT100;
   1:  PR[GP1:91,1] = PR[GP1:90,1] + 57.031;
   1:  PR[GP1:91,2] = PR[GP1:90,2] + 19.670;
   1:L PR[91] 10mm/sec CNT100;
   1:  PR[GP1:91,1] = PR[GP1:90,1] + 54.408;
   1:  PR[GP1:91,2] = PR[GP1:90,2] + 23.737;
   1:L PR[91] 10mm/sec CNT100;
   1:  PR[GP1:91,1] = PR[GP1:90,1] + 51.254;
   1:  PR[GP1:91,2] = PR[GP1:90,2] + 26.827;
   1:L PR[91] 10mm/sec CNT100;
   1:  PR[GP1:91,1] = PR[GP1:90,1] + 46.567;
   1:  PR[GP1:91,2] = PR[GP1:90,2] + 31.068;
   1:L PR[91] 10mm/sec CNT100;
   1:  PR[GP1:91,1] = PR[GP1:90,1] + 42.942;
   1:  PR[GP1:91,2] = PR[GP1:90,2] + 33.342;
   1:L PR[91] 10mm/sec CNT100;
   1:  PR[GP1:91,1] = PR[GP1:90,1] + 36.485;
   1:  PR[GP1:91,2] = PR[GP1:90,2] + 36.164;
   1:L PR[91] 10mm/sec CNT100;
   1:  PR[GP1:91,1] = PR[GP1:90,1] + 32.641;
   1:  PR[GP1:91,2] = PR[GP1:90,2] + 37.566;
   1:L PR[91] 10mm/sec CNT100;
   1:  PR[GP1:91,1] = PR[GP1:90,1] + 29.004;
   1:  PR[GP1:91,2] = PR[GP1:90,2] + 38.082;
   1:L PR[91] 10mm/sec CNT100;
   1:  PR[GP1:91,1] = PR[GP1:90,1] + 21.077;
   1:  PR[GP1:91,2] = PR[GP1:90,2] + 38.818;
   1:L PR[91] 10mm/sec CNT100;
   1:  PR[GP1:91,1] = PR[GP1:90,1] + 17.714;
   1:  PR[GP1:91,2] = PR[GP1:90,2] + 38.595;
   1:L PR[91] 10mm/sec CNT100;
   1:  PR[GP1:91,1] = PR[GP1:90,1] + 9.142;
   1:  PR[GP1:91,2] = PR[GP1:90,2] + 36.571;
   1:L PR[91] 10mm/sec CNT100;
   1:  PR[GP1:91,1] = PR[GP1:90,1] + 6.235;
   1:  PR[GP1:91,2] = PR[GP1:90,2] + 35.735;
   1:L PR[91] 10mm/sec CNT100;
   1:  PR[GP1:91,1] = PR[GP1:90,1] + 5.060;
   1:  PR[GP1:91,2] = PR[GP1:90,2] + 35.119;
   1:L PR[91] 10mm/sec CNT100;
   1:  PR[GP1:91,1] = PR[GP1:90,1] + 3.131;
   1:  PR[GP1:91,2] = PR[GP1:90,2] + 34.077;
   1:L PR[91] 10mm/sec CNT100;
   1:  PR[GP1:91,1] = PR[GP1:90,1] + -0.263;
   1:  PR[GP1:91,2] = PR[GP1:90,2] + 31.317;
   1:L PR[91] 10mm/sec CNT100;
   1:  PR[GP1:91,1] = PR[GP1:90,1] + -3.649;
   1:  PR[GP1:91,2] = PR[GP1:90,2] + 34.069;
   1:L PR[91] 10mm/sec CNT100;
   1:  PR[GP1:91,1] = PR[GP1:90,1] + -5.589;
   1:  PR[GP1:91,2] = PR[GP1:90,2] + 35.120;
   1:L PR[91] 10mm/sec CNT100;
   1:  PR[GP1:91,1] = PR[GP1:90,1] + -6.761;
   1:  PR[GP1:91,2] = PR[GP1:90,2] + 35.736;
   1:L PR[91] 10mm/sec CNT100;
   1:  PR[GP1:91,1] = PR[GP1:90,1] + -9.664;
   1:  PR[GP1:91,2] = PR[GP1:90,2] + 36.571;
   1:L PR[91] 10mm/sec CNT100;
   1:  PR[GP1:91,1] = PR[GP1:90,1] + -18.239;
   1:  PR[GP1:91,2] = PR[GP1:90,2] + 38.595;
   1:L PR[91] 10mm/sec CNT100;
   1:  PR[GP1:91,1] = PR[GP1:90,1] + -21.599;
   1:  PR[GP1:91,2] = PR[GP1:90,2] + 38.817;
   1:L PR[91] 10mm/sec CNT100;
   1:  PR[GP1:91,1] = PR[GP1:90,1] + -25.389;
   1:  PR[GP1:91,2] = PR[GP1:90,2] + 38.292;
   1:L PR[91] 10mm/sec CNT100;
   1:  PR[GP1:91,1] = PR[GP1:90,1] + -33.201;
   1:  PR[GP1:91,2] = PR[GP1:90,2] + 37.558;
   1:L PR[91] 10mm/sec CNT100;
   1:  PR[GP1:91,1] = PR[GP1:90,1] + -37.026;
   1:  PR[GP1:91,2] = PR[GP1:90,2] + 36.157;
   1:L PR[91] 10mm/sec CNT100;
   1:  PR[GP1:91,1] = PR[GP1:90,1] + -43.483;
   1:  PR[GP1:91,2] = PR[GP1:90,2] + 33.334;
   1:L PR[91] 10mm/sec CNT100;
   1:  PR[GP1:91,1] = PR[GP1:90,1] + -47.121;
   1:  PR[GP1:91,2] = PR[GP1:90,2] + 31.040;
   1:L PR[91] 10mm/sec CNT100;
   1:  PR[GP1:91,1] = PR[GP1:90,1] + -50.429;
   1:  PR[GP1:91,2] = PR[GP1:90,2] + 27.811;
   1:L PR[91] 10mm/sec CNT100;
   1:  PR[GP1:91,1] = PR[GP1:90,1] + -54.982;
   1:  PR[GP1:91,2] = PR[GP1:90,2] + 23.688;
   1:L PR[91] 10mm/sec CNT100;
   1:  PR[GP1:91,1] = PR[GP1:90,1] + -57.570;
   1:  PR[GP1:91,2] = PR[GP1:90,2] + 19.649;
   1:L PR[91] 10mm/sec CNT100;
   1:  PR[GP1:91,1] = PR[GP1:90,1] + -60.280;
   1:  PR[GP1:91,2] = PR[GP1:90,2] + 14.754;
   1:L PR[91] 10mm/sec CNT100;
   1:  PR[GP1:91,1] = PR[GP1:90,1] + -61.928;
   1:  PR[GP1:91,2] = PR[GP1:90,2] + 10.212;
   1:L PR[91] 10mm/sec CNT100;
   1:  PR[GP1:91,1] = PR[GP1:90,1] + -62.462;
   1:  PR[GP1:91,2] = PR[GP1:90,2] + 5.442;
   1:L PR[91] 10mm/sec CNT100;
   1:  PR[GP1:91,1] = PR[GP1:90,1] + -63.349;
   1:  PR[GP1:91,2] = PR[GP1:90,2] + 0.261;
   1:L PR[91] 10mm/sec CNT100;
   1:  PR[GP1:91,1] = PR[GP1:90,1] + -62.826;
   1:  PR[GP1:91,2] = PR[GP1:90,2] + -4.438;
   1:L PR[91] 10mm/sec CNT100;
   1:  PR[GP1:91,1] = PR[GP1:90,1] + -61.938;
   1:  PR[GP1:91,2] = PR[GP1:90,2] + -9.627;
   1:L PR[91] 10mm/sec CNT100;
   1:  PR[GP1:91,1] = PR[GP1:90,1] + -60.284;
   1:  PR[GP1:91,2] = PR[GP1:90,2] + -14.185;
   1:L PR[91] 10mm/sec CNT100;
   1:  PR[GP1:91,1] = PR[GP1:90,1] + -57.585;
   1:  PR[GP1:91,2] = PR[GP1:90,2] + -19.071;
   1:L PR[91] 10mm/sec CNT100;
   1:  PR[GP1:91,1] = PR[GP1:90,1] + -54.991;
   1:  PR[GP1:91,2] = PR[GP1:90,2] + -23.120;
   1:L PR[91] 10mm/sec CNT100;
   1:  PR[GP1:91,1] = PR[GP1:90,1] + -51.832;
   1:  PR[GP1:91,2] = PR[GP1:90,2] + -26.220;
   1:L PR[91] 10mm/sec CNT100;
   1:  PR[GP1:91,1] = PR[GP1:90,1] + -47.166;
   1:  PR[GP1:91,2] = PR[GP1:90,2] + -30.453;
   1:L PR[91] 10mm/sec CNT100;
   1:  PR[GP1:91,1] = PR[GP1:90,1] + -43.519;
   1:  PR[GP1:91,2] = PR[GP1:90,2] + -32.752;
   1:L PR[91] 10mm/sec CNT100;
   1:  PR[GP1:91,1] = PR[GP1:90,1] + -37.088;
   1:  PR[GP1:91,2] = PR[GP1:90,2] + -35.583;
   1:L PR[91] 10mm/sec CNT100;
   1:  PR[GP1:91,1] = PR[GP1:90,1] + -33.251;
   1:  PR[GP1:91,2] = PR[GP1:90,2] + -36.988;
   1:L PR[91] 10mm/sec CNT100;
   1:  PR[GP1:91,1] = PR[GP1:90,1] + -29.603;
   1:  PR[GP1:91,2] = PR[GP1:90,2] + -37.507;
   1:L PR[91] 10mm/sec CNT100;
   1:  PR[GP1:91,1] = PR[GP1:90,1] + -21.701;
   1:  PR[GP1:91,2] = PR[GP1:90,2] + -38.265;
   1:L PR[91] 10mm/sec CNT100;
   1:  PR[GP1:91,1] = PR[GP1:90,1] + -18.328;
   1:  PR[GP1:91,2] = PR[GP1:90,2] + -38.043;
   1:L PR[91] 10mm/sec CNT100;
   1:  PR[GP1:91,1] = PR[GP1:90,1] + -9.894;
   1:  PR[GP1:91,2] = PR[GP1:90,2] + -36.113;
   1:L PR[91] 10mm/sec CNT100;
   1:  PR[GP1:91,1] = PR[GP1:90,1] + -6.936;
   1:  PR[GP1:91,2] = PR[GP1:90,2] + -35.264;
   1:L PR[91] 10mm/sec CNT100;
   1:  PR[GP1:91,1] = PR[GP1:90,1] + -0.267;
   1:  PR[GP1:91,2] = PR[GP1:90,2] + -31.356;
   1:L PR[91] 10mm/sec CNT100;
   1:  PR[GP1:91,1] = PR[GP1:90,1] + 6.152;
   1:  PR[GP1:91,2] = PR[GP1:90,2] + -35.332;
   1:  PR[GP1:91,3] = PR[GP1:90,3] + 69.845;
   1:L PR[91] 10mm/sec CNT100;
   1:  PR[GP1:91,1] = PR[GP1:90,1] + 8.993;
   1:  PR[GP1:91,2] = PR[GP1:90,2] + -36.148;
   1:L PR[91] 10mm/sec CNT100;
   1:  PR[GP1:91,1] = PR[GP1:90,1] + 17.626;
   1:  PR[GP1:91,2] = PR[GP1:90,2] + -38.123;
   1:L PR[91] 10mm/sec CNT100;
   1:  PR[GP1:91,1] = PR[GP1:90,1] + 20.853;
   1:  PR[GP1:91,2] = PR[GP1:90,2] + -38.337;
   1:L PR[91] 10mm/sec CNT100;
   1:  PR[GP1:91,1] = PR[GP1:90,1] + 24.493;
   1:  PR[GP1:91,2] = PR[GP1:90,2] + -37.835;
   1:L PR[91] 10mm/sec CNT100;
   1:  PR[GP1:91,1] = PR[GP1:90,1] + 32.499;
   1:  PR[GP1:91,2] = PR[GP1:90,2] + -37.057;
   1:L PR[91] 10mm/sec CNT100;
   1:  PR[GP1:91,1] = PR[GP1:90,1] + 36.202;
   1:  PR[GP1:91,2] = PR[GP1:90,2] + -35.705;
   1:L PR[91] 10mm/sec CNT100;
   1:  PR[GP1:91,1] = PR[GP1:90,1] + 42.833;
   1:  PR[GP1:91,2] = PR[GP1:90,2] + -32.789;
   1:L PR[91] 10mm/sec CNT100;
   1:  PR[GP1:91,1] = PR[GP1:90,1] + 46.338;
   1:  PR[GP1:91,2] = PR[GP1:90,2] + -30.590;
   1:L PR[91] 10mm/sec CNT100;
   1:  PR[GP1:91,1] = PR[GP1:90,1] + 49.539;
   1:  PR[GP1:91,2] = PR[GP1:90,2] + -27.470;
   1:L PR[91] 10mm/sec CNT100;
   1:  PR[GP1:91,1] = PR[GP1:90,1] + 54.243;
   1:  PR[GP1:91,2] = PR[GP1:90,2] + -23.191;
   1:L PR[91] 10mm/sec CNT100;
   1:  PR[GP1:91,1] = PR[GP1:90,1] + 56.784;
   1:  PR[GP1:91,2] = PR[GP1:90,2] + -19.250;
   1:L PR[91] 10mm/sec CNT100;
   1:  PR[GP1:91,1] = PR[GP1:90,1] + 59.591;
   1:  PR[GP1:91,2] = PR[GP1:90,2] + -14.177;
   1:L PR[91] 10mm/sec CNT100;
   1:  PR[GP1:91,1] = PR[GP1:90,1] + 61.187;
   1:  PR[GP1:91,2] = PR[GP1:90,2] + -9.838;
   1:L PR[91] 10mm/sec CNT100;
   1:  PR[GP1:91,1] = PR[GP1:90,1] + 61.725;
   1:  PR[GP1:91,2] = PR[GP1:90,2] + -5.099;
   1:L PR[91] 10mm/sec CNT100;
   1:  PR[GP1:91,1] = PR[GP1:90,1] + 62.645;
   1:  PR[GP1:91,2] = PR[GP1:90,2] + 0.296;
   1:L PR[91] 10mm/sec CNT100;
   1:  PR[GP1:91,1] = PR[GP1:90,1] + 62.117;
   1:  PR[GP1:91,2] = PR[GP1:90,2] + 4.968;
   1:L PR[91] 10mm/sec CNT100;
   1:  PR[GP1:91,1] = PR[GP1:90,1] + 61.189;
   1:  PR[GP1:91,2] = PR[GP1:90,2] + 10.391;
   1:L PR[91] 10mm/sec CNT100;
   1:  PR[GP1:91,1] = PR[GP1:90,1] + 59.587;
   1:  PR[GP1:91,2] = PR[GP1:90,2] + 14.746;
   1:L PR[91] 10mm/sec CNT100;
   1:  PR[GP1:91,1] = PR[GP1:90,1] + 56.768;
   1:  PR[GP1:91,2] = PR[GP1:90,2] + 19.828;
   1:L PR[91] 10mm/sec CNT100;
   1:  PR[GP1:91,1] = PR[GP1:90,1] + 54.221;
   1:  PR[GP1:91,2] = PR[GP1:90,2] + 23.779;
   1:L PR[91] 10mm/sec CNT100;
   1:  PR[GP1:91,1] = PR[GP1:90,1] + 51.156;
   1:  PR[GP1:91,2] = PR[GP1:90,2] + 26.781;
   1:L PR[91] 10mm/sec CNT100;
   1:  PR[GP1:91,1] = PR[GP1:90,1] + 46.310;
   1:  PR[GP1:91,2] = PR[GP1:90,2] + 31.166;
   1:L PR[91] 10mm/sec CNT100;
   1:  PR[GP1:91,1] = PR[GP1:90,1] + 42.796;
   1:  PR[GP1:91,2] = PR[GP1:90,2] + 33.371;
   1:L PR[91] 10mm/sec CNT100;
   1:  PR[GP1:91,1] = PR[GP1:90,1] + 36.139;
   1:  PR[GP1:91,2] = PR[GP1:90,2] + 36.280;
   1:L PR[91] 10mm/sec CNT100;
   1:  PR[GP1:91,1] = PR[GP1:90,1] + 32.422;
   1:  PR[GP1:91,2] = PR[GP1:90,2] + 37.636;
   1:L PR[91] 10mm/sec CNT100;
   1:  PR[GP1:91,1] = PR[GP1:90,1] + 28.905;
   1:  PR[GP1:91,2] = PR[GP1:90,2] + 38.135;
   1:L PR[91] 10mm/sec CNT100;
   1:  PR[GP1:91,1] = PR[GP1:90,1] + 20.775;
   1:  PR[GP1:91,2] = PR[GP1:90,2] + 38.890;
   1:L PR[91] 10mm/sec CNT100;
   1:  PR[GP1:91,1] = PR[GP1:90,1] + 17.535;
   1:  PR[GP1:91,2] = PR[GP1:90,2] + 38.675;
   1:L PR[91] 10mm/sec CNT100;
   1:  PR[GP1:91,1] = PR[GP1:90,1] + 8.761;
   1:  PR[GP1:91,2] = PR[GP1:90,2] + 36.603;
   1:L PR[91] 10mm/sec CNT100;
   1:  PR[GP1:91,1] = PR[GP1:90,1] + 5.977;
   1:  PR[GP1:91,2] = PR[GP1:90,2] + 35.802;
   1:L PR[91] 10mm/sec CNT100;
   1:  PR[GP1:91,1] = PR[GP1:90,1] + 4.775;
   1:  PR[GP1:91,2] = PR[GP1:90,2] + 35.172;
   1:L PR[91] 10mm/sec CNT100;
   1:  PR[GP1:91,1] = PR[GP1:90,1] + 2.958;
   1:  PR[GP1:91,2] = PR[GP1:90,2] + 34.191;
   1:L PR[91] 10mm/sec CNT100;
   1:  PR[GP1:91,1] = PR[GP1:90,1] + -0.263;
   1:  PR[GP1:91,2] = PR[GP1:90,2] + 31.571;
   1:L PR[91] 10mm/sec CNT100;
   1:  PR[GP1:91,1] = PR[GP1:90,1] + -3.477;
   1:  PR[GP1:91,2] = PR[GP1:90,2] + 34.184;
   1:L PR[91] 10mm/sec CNT100;
   1:  PR[GP1:91,1] = PR[GP1:90,1] + -5.303;
   1:  PR[GP1:91,2] = PR[GP1:90,2] + 35.173;
   1:L PR[91] 10mm/sec CNT100;
   1:  PR[GP1:91,1] = PR[GP1:90,1] + -6.503;
   1:  PR[GP1:91,2] = PR[GP1:90,2] + 35.804;
   1:L PR[91] 10mm/sec CNT100;
   1:  PR[GP1:91,1] = PR[GP1:90,1] + -9.283;
   1:  PR[GP1:91,2] = PR[GP1:90,2] + 36.603;
   1:L PR[91] 10mm/sec CNT100;
   1:  PR[GP1:91,1] = PR[GP1:90,1] + -18.060;
   1:  PR[GP1:91,2] = PR[GP1:90,2] + 38.675;
   1:L PR[91] 10mm/sec CNT100;
   1:  PR[GP1:91,1] = PR[GP1:90,1] + -21.296;
   1:  PR[GP1:91,2] = PR[GP1:90,2] + 38.889;
   1:L PR[91] 10mm/sec CNT100;
   1:  PR[GP1:91,1] = PR[GP1:90,1] + -24.950;
   1:  PR[GP1:91,2] = PR[GP1:90,2] + 38.383;
   1:L PR[91] 10mm/sec CNT100;
   1:  PR[GP1:91,1] = PR[GP1:90,1] + -32.981;
   1:  PR[GP1:91,2] = PR[GP1:90,2] + 37.628;
   1:L PR[91] 10mm/sec CNT100;
   1:  PR[GP1:91,1] = PR[GP1:90,1] + -36.680;
   1:  PR[GP1:91,2] = PR[GP1:90,2] + 36.273;
   1:L PR[91] 10mm/sec CNT100;
   1:  PR[GP1:91,1] = PR[GP1:90,1] + -43.336;
   1:  PR[GP1:91,2] = PR[GP1:90,2] + 33.363;
   1:L PR[91] 10mm/sec CNT100;
   1:  PR[GP1:91,1] = PR[GP1:90,1] + -46.863;
   1:  PR[GP1:91,2] = PR[GP1:90,2] + 31.139;
   1:L PR[91] 10mm/sec CNT100;
   1:  PR[GP1:91,1] = PR[GP1:90,1] + -50.071;
   1:  PR[GP1:91,2] = PR[GP1:90,2] + 28.007;
   1:L PR[91] 10mm/sec CNT100;
   1:  PR[GP1:91,1] = PR[GP1:90,1] + -54.793;
   1:  PR[GP1:91,2] = PR[GP1:90,2] + 23.732;
   1:L PR[91] 10mm/sec CNT100;
   1:  PR[GP1:91,1] = PR[GP1:90,1] + -57.307;
   1:  PR[GP1:91,2] = PR[GP1:90,2] + 19.808;
   1:L PR[91] 10mm/sec CNT100;
   1:  PR[GP1:91,1] = PR[GP1:90,1] + -60.125;
   1:  PR[GP1:91,2] = PR[GP1:90,2] + 14.718;
   1:L PR[91] 10mm/sec CNT100;
   1:  PR[GP1:91,1] = PR[GP1:90,1] + -61.728;
   1:  PR[GP1:91,2] = PR[GP1:90,2] + 10.302;
   1:L PR[91] 10mm/sec CNT100;
   1:  PR[GP1:91,1] = PR[GP1:90,1] + -62.248;
   1:  PR[GP1:91,2] = PR[GP1:90,2] + 5.663;
   1:L PR[91] 10mm/sec CNT100;
   1:  PR[GP1:91,1] = PR[GP1:90,1] + -63.172;
   1:  PR[GP1:91,2] = PR[GP1:90,2] + 0.261;
   1:L PR[91] 10mm/sec CNT100;
   1:  PR[GP1:91,1] = PR[GP1:90,1] + -62.663;
   1:  PR[GP1:91,2] = PR[GP1:90,2] + -4.310;
   1:L PR[91] 10mm/sec CNT100;
   1:  PR[GP1:91,1] = PR[GP1:90,1] + -61.738;
   1:  PR[GP1:91,2] = PR[GP1:90,2] + -9.716;
   1:L PR[91] 10mm/sec CNT100;
   1:  PR[GP1:91,1] = PR[GP1:90,1] + -60.129;
   1:  PR[GP1:91,2] = PR[GP1:90,2] + -14.149;
   1:L PR[91] 10mm/sec CNT100;
   1:  PR[GP1:91,1] = PR[GP1:90,1] + -57.323;
   1:  PR[GP1:91,2] = PR[GP1:90,2] + -19.230;
   1:L PR[91] 10mm/sec CNT100;
   1:  PR[GP1:91,1] = PR[GP1:90,1] + -54.803;
   1:  PR[GP1:91,2] = PR[GP1:90,2] + -23.163;
   1:L PR[91] 10mm/sec CNT100;
   1:  PR[GP1:91,1] = PR[GP1:90,1] + -51.734;
   1:  PR[GP1:91,2] = PR[GP1:90,2] + -26.174;
   1:L PR[91] 10mm/sec CNT100;
   1:  PR[GP1:91,1] = PR[GP1:90,1] + -46.909;
   1:  PR[GP1:91,2] = PR[GP1:90,2] + -30.551;
   1:L PR[91] 10mm/sec CNT100;
   1:  PR[GP1:91,1] = PR[GP1:90,1] + -43.374;
   1:  PR[GP1:91,2] = PR[GP1:90,2] + -32.781;
   1:L PR[91] 10mm/sec CNT100;
   1:  PR[GP1:91,1] = PR[GP1:90,1] + -36.743;
   1:  PR[GP1:91,2] = PR[GP1:90,2] + -35.699;
   1:L PR[91] 10mm/sec CNT100;
   1:  PR[GP1:91,1] = PR[GP1:90,1] + -33.033;
   1:  PR[GP1:91,2] = PR[GP1:90,2] + -37.058;
   1:L PR[91] 10mm/sec CNT100;
   1:  PR[GP1:91,1] = PR[GP1:90,1] + -29.505;
   1:  PR[GP1:91,2] = PR[GP1:90,2] + -37.560;
   1:L PR[91] 10mm/sec CNT100;
   1:  PR[GP1:91,1] = PR[GP1:90,1] + -21.401;
   1:  PR[GP1:91,2] = PR[GP1:90,2] + -38.337;
   1:L PR[91] 10mm/sec CNT100;
   1:  PR[GP1:91,1] = PR[GP1:90,1] + -18.151;
   1:  PR[GP1:91,2] = PR[GP1:90,2] + -38.123;
   1:L PR[91] 10mm/sec CNT100;
   1:  PR[GP1:91,1] = PR[GP1:90,1] + -9.519;
   1:  PR[GP1:91,2] = PR[GP1:90,2] + -36.148;
   1:L PR[91] 10mm/sec CNT100;
   1:  PR[GP1:91,1] = PR[GP1:90,1] + -6.682;
   1:  PR[GP1:91,2] = PR[GP1:90,2] + -35.333;
   1:L PR[91] 10mm/sec CNT100;
   1:  PR[GP1:91,1] = PR[GP1:90,1] + -0.266;
   1:  PR[GP1:91,2] = PR[GP1:90,2] + -31.575;
   1:L PR[91] 10mm/sec CNT100;
   1:  PR[GP1:91,1] = PR[GP1:90,1] + 5.898;
   1:  PR[GP1:91,2] = PR[GP1:90,2] + -35.401;
   1:  PR[GP1:91,3] = PR[GP1:90,3] + 70.455;
   1:L PR[91] 10mm/sec CNT100;
   1:  PR[GP1:91,1] = PR[GP1:90,1] + 8.618;
   1:  PR[GP1:91,2] = PR[GP1:90,2] + -36.182;
   1:L PR[91] 10mm/sec CNT100;
   1:  PR[GP1:91,1] = PR[GP1:90,1] + 17.449;
   1:  PR[GP1:91,2] = PR[GP1:90,2] + -38.203;
   1:L PR[91] 10mm/sec CNT100;
   1:  PR[GP1:91,1] = PR[GP1:90,1] + 20.553;
   1:  PR[GP1:91,2] = PR[GP1:90,2] + -38.409;
   1:L PR[91] 10mm/sec CNT100;
   1:  PR[GP1:91,1] = PR[GP1:90,1] + 24.057;
   1:  PR[GP1:91,2] = PR[GP1:90,2] + -37.926;
   1:L PR[91] 10mm/sec CNT100;
   1:  PR[GP1:91,1] = PR[GP1:90,1] + 32.282;
   1:  PR[GP1:91,2] = PR[GP1:90,2] + -37.126;
   1:L PR[91] 10mm/sec CNT100;
   1:  PR[GP1:91,1] = PR[GP1:90,1] + 35.857;
   1:  PR[GP1:91,2] = PR[GP1:90,2] + -35.821;
   1:L PR[91] 10mm/sec CNT100;
   1:  PR[GP1:91,1] = PR[GP1:90,1] + 42.688;
   1:  PR[GP1:91,2] = PR[GP1:90,2] + -32.817;
   1:L PR[91] 10mm/sec CNT100;
   1:  PR[GP1:91,1] = PR[GP1:90,1] + 46.082;
   1:  PR[GP1:91,2] = PR[GP1:90,2] + -30.688;
   1:L PR[91] 10mm/sec CNT100;
   1:  PR[GP1:91,1] = PR[GP1:90,1] + 49.184;
   1:  PR[GP1:91,2] = PR[GP1:90,2] + -27.665;
   1:L PR[91] 10mm/sec CNT100;
   1:  PR[GP1:91,1] = PR[GP1:90,1] + 54.056;
   1:  PR[GP1:91,2] = PR[GP1:90,2] + -23.233;
   1:L PR[91] 10mm/sec CNT100;
   1:  PR[GP1:91,1] = PR[GP1:90,1] + 56.523;
   1:  PR[GP1:91,2] = PR[GP1:90,2] + -19.407;
   1:L PR[91] 10mm/sec CNT100;
   1:  PR[GP1:91,1] = PR[GP1:90,1] + 59.437;
   1:  PR[GP1:91,2] = PR[GP1:90,2] + -14.140;
   1:L PR[91] 10mm/sec CNT100;
   1:  PR[GP1:91,1] = PR[GP1:90,1] + 60.987;
   1:  PR[GP1:91,2] = PR[GP1:90,2] + -9.925;
   1:L PR[91] 10mm/sec CNT100;
   1:  PR[GP1:91,1] = PR[GP1:90,1] + 61.511;
   1:  PR[GP1:91,2] = PR[GP1:90,2] + -5.318;
   1:L PR[91] 10mm/sec CNT100;
   1:  PR[GP1:91,1] = PR[GP1:90,1] + 62.468;
   1:  PR[GP1:91,2] = PR[GP1:90,2] + 0.296;
   1:L PR[91] 10mm/sec CNT100;
   1:  PR[GP1:91,1] = PR[GP1:90,1] + 61.955;
   1:  PR[GP1:91,2] = PR[GP1:90,2] + 4.837;
   1:L PR[91] 10mm/sec CNT100;
   1:  PR[GP1:91,1] = PR[GP1:90,1] + 60.989;
   1:  PR[GP1:91,2] = PR[GP1:90,2] + 10.478;
   1:L PR[91] 10mm/sec CNT100;
   1:  PR[GP1:91,1] = PR[GP1:90,1] + 59.433;
   1:  PR[GP1:91,2] = PR[GP1:90,2] + 14.710;
   1:L PR[91] 10mm/sec CNT100;
   1:  PR[GP1:91,1] = PR[GP1:90,1] + 56.506;
   1:  PR[GP1:91,2] = PR[GP1:90,2] + 19.987;
   1:L PR[91] 10mm/sec CNT100;
   1:  PR[GP1:91,1] = PR[GP1:90,1] + 54.033;
   1:  PR[GP1:91,2] = PR[GP1:90,2] + 23.822;
   1:L PR[91] 10mm/sec CNT100;
   1:  PR[GP1:91,1] = PR[GP1:90,1] + 51.059;
   1:  PR[GP1:91,2] = PR[GP1:90,2] + 26.735;
   1:L PR[91] 10mm/sec CNT100;
   1:  PR[GP1:91,1] = PR[GP1:90,1] + 46.053;
   1:  PR[GP1:91,2] = PR[GP1:90,2] + 31.265;
   1:L PR[91] 10mm/sec CNT100;
   1:  PR[GP1:91,1] = PR[GP1:90,1] + 42.649;
   1:  PR[GP1:91,2] = PR[GP1:90,2] + 33.400;
   1:L PR[91] 10mm/sec CNT100;
   1:  PR[GP1:91,1] = PR[GP1:90,1] + 35.793;
   1:  PR[GP1:91,2] = PR[GP1:90,2] + 36.396;
   1:L PR[91] 10mm/sec CNT100;
   1:  PR[GP1:91,1] = PR[GP1:90,1] + 32.203;
   1:  PR[GP1:91,2] = PR[GP1:90,2] + 37.706;
   1:L PR[91] 10mm/sec CNT100;
   1:  PR[GP1:91,1] = PR[GP1:90,1] + 28.806;
   1:  PR[GP1:91,2] = PR[GP1:90,2] + 38.188;
   1:L PR[91] 10mm/sec CNT100;
   1:  PR[GP1:91,1] = PR[GP1:90,1] + 20.473;
   1:  PR[GP1:91,2] = PR[GP1:90,2] + 38.962;
   1:L PR[91] 10mm/sec CNT100;
   1:  PR[GP1:91,1] = PR[GP1:90,1] + 17.357;
   1:  PR[GP1:91,2] = PR[GP1:90,2] + 38.755;
   1:L PR[91] 10mm/sec CNT100;
   1:  PR[GP1:91,1] = PR[GP1:90,1] + 8.381;
   1:  PR[GP1:91,2] = PR[GP1:90,2] + 36.635;
   1:L PR[91] 10mm/sec CNT100;
   1:  PR[GP1:91,1] = PR[GP1:90,1] + 5.719;
   1:  PR[GP1:91,2] = PR[GP1:90,2] + 35.870;
   1:L PR[91] 10mm/sec CNT100;
   1:  PR[GP1:91,1] = PR[GP1:90,1] + 4.490;
   1:  PR[GP1:91,2] = PR[GP1:90,2] + 35.226;
   1:L PR[91] 10mm/sec CNT100;
   1:  PR[GP1:91,1] = PR[GP1:90,1] + 2.785;
   1:  PR[GP1:91,2] = PR[GP1:90,2] + 34.305;
   1:L PR[91] 10mm/sec CNT100;
   1:  PR[GP1:91,1] = PR[GP1:90,1] + -0.263;
   1:  PR[GP1:91,2] = PR[GP1:90,2] + 31.826;
   1:L PR[91] 10mm/sec CNT100;
   1:  PR[GP1:91,1] = PR[GP1:90,1] + -3.304;
   1:  PR[GP1:91,2] = PR[GP1:90,2] + 34.298;
   1:L PR[91] 10mm/sec CNT100;
   1:  PR[GP1:91,1] = PR[GP1:90,1] + -5.019;
   1:  PR[GP1:91,2] = PR[GP1:90,2] + 35.227;
   1:L PR[91] 10mm/sec CNT100;
   1:  PR[GP1:91,1] = PR[GP1:90,1] + -6.244;
   1:  PR[GP1:91,2] = PR[GP1:90,2] + 35.871;
   1:L PR[91] 10mm/sec CNT100;
   1:  PR[GP1:91,1] = PR[GP1:90,1] + -8.903;
   1:  PR[GP1:91,2] = PR[GP1:90,2] + 36.636;
   1:L PR[91] 10mm/sec CNT100;
   1:  PR[GP1:91,1] = PR[GP1:90,1] + -17.881;
   1:  PR[GP1:91,2] = PR[GP1:90,2] + 38.755;
   1:L PR[91] 10mm/sec CNT100;
   1:  PR[GP1:91,1] = PR[GP1:90,1] + -20.994;
   1:  PR[GP1:91,2] = PR[GP1:90,2] + 38.960;
   1:L PR[91] 10mm/sec CNT100;
   1:  PR[GP1:91,1] = PR[GP1:90,1] + -24.510;
   1:  PR[GP1:91,2] = PR[GP1:90,2] + 38.474;
   1:L PR[91] 10mm/sec CNT100;
   1:  PR[GP1:91,1] = PR[GP1:90,1] + -32.761;
   1:  PR[GP1:91,2] = PR[GP1:90,2] + 37.698;
   1:L PR[91] 10mm/sec CNT100;
   1:  PR[GP1:91,1] = PR[GP1:90,1] + -36.333;
   1:  PR[GP1:91,2] = PR[GP1:90,2] + 36.390;
   1:L PR[91] 10mm/sec CNT100;
   1:  PR[GP1:91,1] = PR[GP1:90,1] + -43.189;
   1:  PR[GP1:91,2] = PR[GP1:90,2] + 33.392;
   1:L PR[91] 10mm/sec CNT100;
   1:  PR[GP1:91,1] = PR[GP1:90,1] + -46.605;
   1:  PR[GP1:91,2] = PR[GP1:90,2] + 31.239;
   1:L PR[91] 10mm/sec CNT100;
   1:  PR[GP1:91,1] = PR[GP1:90,1] + -49.714;
   1:  PR[GP1:91,2] = PR[GP1:90,2] + 28.204;
   1:L PR[91] 10mm/sec CNT100;
   1:  PR[GP1:91,1] = PR[GP1:90,1] + -54.605;
   1:  PR[GP1:91,2] = PR[GP1:90,2] + 23.776;
   1:L PR[91] 10mm/sec CNT100;
   1:  PR[GP1:91,1] = PR[GP1:90,1] + -57.044;
   1:  PR[GP1:91,2] = PR[GP1:90,2] + 19.968;
   1:L PR[91] 10mm/sec CNT100;
   1:  PR[GP1:91,1] = PR[GP1:90,1] + -59.971;
   1:  PR[GP1:91,2] = PR[GP1:90,2] + 14.682;
   1:L PR[91] 10mm/sec CNT100;
   1:  PR[GP1:91,1] = PR[GP1:90,1] + -61.528;
   1:  PR[GP1:91,2] = PR[GP1:90,2] + 10.392;
   1:L PR[91] 10mm/sec CNT100;
   1:  PR[GP1:91,1] = PR[GP1:90,1] + -62.033;
   1:  PR[GP1:91,2] = PR[GP1:90,2] + 5.883;
   1:L PR[91] 10mm/sec CNT100;
   1:  PR[GP1:91,1] = PR[GP1:90,1] + -62.995;
   1:  PR[GP1:91,2] = PR[GP1:90,2] + 0.261;
   1:L PR[91] 10mm/sec CNT100;
   1:  PR[GP1:91,1] = PR[GP1:90,1] + -62.500;
   1:  PR[GP1:91,2] = PR[GP1:90,2] + -4.182;
   1:L PR[91] 10mm/sec CNT100;
   1:  PR[GP1:91,1] = PR[GP1:90,1] + -61.538;
   1:  PR[GP1:91,2] = PR[GP1:90,2] + -9.805;
   1:L PR[91] 10mm/sec CNT100;
   1:  PR[GP1:91,1] = PR[GP1:90,1] + -59.975;
   1:  PR[GP1:91,2] = PR[GP1:90,2] + -14.112;
   1:L PR[91] 10mm/sec CNT100;
   1:  PR[GP1:91,1] = PR[GP1:90,1] + -57.061;
   1:  PR[GP1:91,2] = PR[GP1:90,2] + -19.388;
   1:L PR[91] 10mm/sec CNT100;
   1:  PR[GP1:91,1] = PR[GP1:90,1] + -54.615;
   1:  PR[GP1:91,2] = PR[GP1:90,2] + -23.206;
   1:L PR[91] 10mm/sec CNT100;
   1:  PR[GP1:91,1] = PR[GP1:90,1] + -51.636;
   1:  PR[GP1:91,2] = PR[GP1:90,2] + -26.129;
   1:L PR[91] 10mm/sec CNT100;
   1:  PR[GP1:91,1] = PR[GP1:90,1] + -46.653;
   1:  PR[GP1:91,2] = PR[GP1:90,2] + -30.650;
   1:L PR[91] 10mm/sec CNT100;
   1:  PR[GP1:91,1] = PR[GP1:90,1] + -43.228;
   1:  PR[GP1:91,2] = PR[GP1:90,2] + -32.809;
   1:L PR[91] 10mm/sec CNT100;
   1:  PR[GP1:91,1] = PR[GP1:90,1] + -36.398;
   1:  PR[GP1:91,2] = PR[GP1:90,2] + -35.815;
   1:L PR[91] 10mm/sec CNT100;
   1:  PR[GP1:91,1] = PR[GP1:90,1] + -32.815;
   1:  PR[GP1:91,2] = PR[GP1:90,2] + -37.128;
   1:L PR[91] 10mm/sec CNT100;
   1:  PR[GP1:91,1] = PR[GP1:90,1] + -29.407;
   1:  PR[GP1:91,2] = PR[GP1:90,2] + -37.612;
   1:L PR[91] 10mm/sec CNT100;
   1:  PR[GP1:91,1] = PR[GP1:90,1] + -21.101;
   1:  PR[GP1:91,2] = PR[GP1:90,2] + -38.409;
   1:L PR[91] 10mm/sec CNT100;
   1:  PR[GP1:91,1] = PR[GP1:90,1] + -17.974;
   1:  PR[GP1:91,2] = PR[GP1:90,2] + -38.203;
   1:L PR[91] 10mm/sec CNT100;
   1:  PR[GP1:91,1] = PR[GP1:90,1] + -9.143;
   1:  PR[GP1:91,2] = PR[GP1:90,2] + -36.183;
   1:L PR[91] 10mm/sec CNT100;
   1:  PR[GP1:91,1] = PR[GP1:90,1] + -6.427;
   1:  PR[GP1:91,2] = PR[GP1:90,2] + -35.402;
   1:L PR[91] 10mm/sec CNT100;
   1:  PR[GP1:91,1] = PR[GP1:90,1] + -0.266;
   1:  PR[GP1:91,2] = PR[GP1:90,2] + -31.793;
   1:L PR[91] 10mm/sec CNT100;
   1:  PR[GP1:91,1] = PR[GP1:90,1] + 5.643;
   1:  PR[GP1:91,2] = PR[GP1:90,2] + -35.471;
   1:  PR[GP1:91,3] = PR[GP1:90,3] + 71.065;
   1:L PR[91] 10mm/sec CNT100;
   1:  PR[GP1:91,1] = PR[GP1:90,1] + 8.243;
   1:  PR[GP1:91,2] = PR[GP1:90,2] + -36.217;
   1:L PR[91] 10mm/sec CNT100;
   1:  PR[GP1:91,1] = PR[GP1:90,1] + 17.272;
   1:  PR[GP1:91,2] = PR[GP1:90,2] + -38.283;
   1:L PR[91] 10mm/sec CNT100;
   1:  PR[GP1:91,1] = PR[GP1:90,1] + 20.253;
   1:  PR[GP1:91,2] = PR[GP1:90,2] + -38.481;
   1:L PR[91] 10mm/sec CNT100;
   1:  PR[GP1:91,1] = PR[GP1:90,1] + 23.621;
   1:  PR[GP1:91,2] = PR[GP1:90,2] + -38.016;
   1:L PR[91] 10mm/sec CNT100;
   1:  PR[GP1:91,1] = PR[GP1:90,1] + 32.064;
   1:  PR[GP1:91,2] = PR[GP1:90,2] + -37.196;
   1:L PR[91] 10mm/sec CNT100;
   1:  PR[GP1:91,1] = PR[GP1:90,1] + 35.513;
   1:  PR[GP1:91,2] = PR[GP1:90,2] + -35.937;
   1:L PR[91] 10mm/sec CNT100;
   1:  PR[GP1:91,1] = PR[GP1:90,1] + 42.543;
   1:  PR[GP1:91,2] = PR[GP1:90,2] + -32.846;
   1:L PR[91] 10mm/sec CNT100;
   1:  PR[GP1:91,1] = PR[GP1:90,1] + 45.827;
   1:  PR[GP1:91,2] = PR[GP1:90,2] + -30.785;
   1:L PR[91] 10mm/sec CNT100;
   1:  PR[GP1:91,1] = PR[GP1:90,1] + 48.829;
   1:  PR[GP1:91,2] = PR[GP1:90,2] + -27.859;
   1:L PR[91] 10mm/sec CNT100;
   1:  PR[GP1:91,1] = PR[GP1:90,1] + 53.870;
   1:  PR[GP1:91,2] = PR[GP1:90,2] + -23.274;
   1:L PR[91] 10mm/sec CNT100;
   1:  PR[GP1:91,1] = PR[GP1:90,1] + 56.261;
   1:  PR[GP1:91,2] = PR[GP1:90,2] + -19.565;
   1:L PR[91] 10mm/sec CNT100;
   1:  PR[GP1:91,1] = PR[GP1:90,1] + 59.283;
   1:  PR[GP1:91,2] = PR[GP1:90,2] + -14.103;
   1:L PR[91] 10mm/sec CNT100;
   1:  PR[GP1:91,1] = PR[GP1:90,1] + 60.788;
   1:  PR[GP1:91,2] = PR[GP1:90,2] + -10.011;
   1:L PR[91] 10mm/sec CNT100;
   1:  PR[GP1:91,1] = PR[GP1:90,1] + 61.296;
   1:  PR[GP1:91,2] = PR[GP1:90,2] + -5.538;
   1:L PR[91] 10mm/sec CNT100;
   1:  PR[GP1:91,1] = PR[GP1:90,1] + 62.291;
   1:  PR[GP1:91,2] = PR[GP1:90,2] + 0.296;
   1:L PR[91] 10mm/sec CNT100;
   1:  PR[GP1:91,1] = PR[GP1:90,1] + 61.792;
   1:  PR[GP1:91,2] = PR[GP1:90,2] + 4.706;
   1:L PR[91] 10mm/sec CNT100;
   1:  PR[GP1:91,1] = PR[GP1:90,1] + 60.789;
   1:  PR[GP1:91,2] = PR[GP1:90,2] + 10.565;
   1:L PR[91] 10mm/sec CNT100;
   1:  PR[GP1:91,1] = PR[GP1:90,1] + 59.278;
   1:  PR[GP1:91,2] = PR[GP1:90,2] + 14.674;
   1:L PR[91] 10mm/sec CNT100;
   1:  PR[GP1:91,1] = PR[GP1:90,1] + 56.244;
   1:  PR[GP1:91,2] = PR[GP1:90,2] + 20.145;
   1:L PR[91] 10mm/sec CNT100;
   1:  PR[GP1:91,1] = PR[GP1:90,1] + 53.846;
   1:  PR[GP1:91,2] = PR[GP1:90,2] + 23.864;
   1:L PR[91] 10mm/sec CNT100;
   1:  PR[GP1:91,1] = PR[GP1:90,1] + 50.961;
   1:  PR[GP1:91,2] = PR[GP1:90,2] + 26.689;
   1:L PR[91] 10mm/sec CNT100;
   1:  PR[GP1:91,1] = PR[GP1:90,1] + 45.797;
   1:  PR[GP1:91,2] = PR[GP1:90,2] + 31.363;
   1:L PR[91] 10mm/sec CNT100;
   1:  PR[GP1:91,1] = PR[GP1:90,1] + 42.503;
   1:  PR[GP1:91,2] = PR[GP1:90,2] + 33.429;
   1:L PR[91] 10mm/sec CNT100;
   1:  PR[GP1:91,1] = PR[GP1:90,1] + 35.447;
   1:  PR[GP1:91,2] = PR[GP1:90,2] + 36.513;
   1:L PR[91] 10mm/sec CNT100;
   1:  PR[GP1:91,1] = PR[GP1:90,1] + 31.984;
   1:  PR[GP1:91,2] = PR[GP1:90,2] + 37.776;
   1:L PR[91] 10mm/sec CNT100;
   1:  PR[GP1:91,1] = PR[GP1:90,1] + 28.707;
   1:  PR[GP1:91,2] = PR[GP1:90,2] + 38.241;
   1:L PR[91] 10mm/sec CNT100;
   1:  PR[GP1:91,1] = PR[GP1:90,1] + 20.170;
   1:  PR[GP1:91,2] = PR[GP1:90,2] + 39.034;
   1:L PR[91] 10mm/sec CNT100;
   1:  PR[GP1:91,1] = PR[GP1:90,1] + 17.178;
   1:  PR[GP1:91,2] = PR[GP1:90,2] + 38.835;
   1:L PR[91] 10mm/sec CNT100;
   1:  PR[GP1:91,1] = PR[GP1:90,1] + 8.000;
   1:  PR[GP1:91,2] = PR[GP1:90,2] + 36.668;
   1:L PR[91] 10mm/sec CNT100;
   1:  PR[GP1:91,1] = PR[GP1:90,1] + 5.462;
   1:  PR[GP1:91,2] = PR[GP1:90,2] + 35.938;
   1:L PR[91] 10mm/sec CNT100;
   1:  PR[GP1:91,1] = PR[GP1:90,1] + 2.611;
   1:  PR[GP1:91,2] = PR[GP1:90,2] + 34.418;
   1:L PR[91] 10mm/sec CNT100;
   1:  PR[GP1:91,1] = PR[GP1:90,1] + -0.263;
   1:  PR[GP1:91,2] = PR[GP1:90,2] + 32.081;
   1:L PR[91] 10mm/sec CNT100;
   1:  PR[GP1:91,1] = PR[GP1:90,1] + -3.132;
   1:  PR[GP1:91,2] = PR[GP1:90,2] + 34.413;
   1:L PR[91] 10mm/sec CNT100;
   1:  PR[GP1:91,1] = PR[GP1:90,1] + -4.734;
   1:  PR[GP1:91,2] = PR[GP1:90,2] + 35.280;
   1:L PR[91] 10mm/sec CNT100;
   1:  PR[GP1:91,1] = PR[GP1:90,1] + -5.986;
   1:  PR[GP1:91,2] = PR[GP1:90,2] + 35.939;
   1:L PR[91] 10mm/sec CNT100;
   1:  PR[GP1:91,1] = PR[GP1:90,1] + -8.522;
   1:  PR[GP1:91,2] = PR[GP1:90,2] + 36.668;
   1:L PR[91] 10mm/sec CNT100;
   1:  PR[GP1:91,1] = PR[GP1:90,1] + -17.702;
   1:  PR[GP1:91,2] = PR[GP1:90,2] + 38.835;
   1:L PR[91] 10mm/sec CNT100;
   1:  PR[GP1:91,1] = PR[GP1:90,1] + -20.691;
   1:  PR[GP1:91,2] = PR[GP1:90,2] + 39.032;
   1:L PR[91] 10mm/sec CNT100;
   1:  PR[GP1:91,1] = PR[GP1:90,1] + -24.071;
   1:  PR[GP1:91,2] = PR[GP1:90,2] + 38.565;
   1:L PR[91] 10mm/sec CNT100;
   1:  PR[GP1:91,1] = PR[GP1:90,1] + -32.541;
   1:  PR[GP1:91,2] = PR[GP1:90,2] + 37.768;
   1:L PR[91] 10mm/sec CNT100;
   1:  PR[GP1:91,1] = PR[GP1:90,1] + -35.987;
   1:  PR[GP1:91,2] = PR[GP1:90,2] + 36.506;
   1:L PR[91] 10mm/sec CNT100;
   1:  PR[GP1:91,1] = PR[GP1:90,1] + -43.043;
   1:  PR[GP1:91,2] = PR[GP1:90,2] + 33.421;
   1:L PR[91] 10mm/sec CNT100;
   1:  PR[GP1:91,1] = PR[GP1:90,1] + -46.347;
   1:  PR[GP1:91,2] = PR[GP1:90,2] + 31.338;
   1:L PR[91] 10mm/sec CNT100;
   1:  PR[GP1:91,1] = PR[GP1:90,1] + -49.356;
   1:  PR[GP1:91,2] = PR[GP1:90,2] + 28.401;
   1:L PR[91] 10mm/sec CNT100;
   1:  PR[GP1:91,1] = PR[GP1:90,1] + -54.416;
   1:  PR[GP1:91,2] = PR[GP1:90,2] + 23.819;
   1:L PR[91] 10mm/sec CNT100;
   1:  PR[GP1:91,1] = PR[GP1:90,1] + -56.782;
   1:  PR[GP1:91,2] = PR[GP1:90,2] + 20.127;
   1:L PR[91] 10mm/sec CNT100;
   1:  PR[GP1:91,1] = PR[GP1:90,1] + -59.816;
   1:  PR[GP1:91,2] = PR[GP1:90,2] + 14.646;
   1:L PR[91] 10mm/sec CNT100;
   1:  PR[GP1:91,1] = PR[GP1:90,1] + -61.327;
   1:  PR[GP1:91,2] = PR[GP1:90,2] + 10.481;
   1:L PR[91] 10mm/sec CNT100;
   1:  PR[GP1:91,1] = PR[GP1:90,1] + -61.818;
   1:  PR[GP1:91,2] = PR[GP1:90,2] + 6.103;
   1:L PR[91] 10mm/sec CNT100;
   1:  PR[GP1:91,1] = PR[GP1:90,1] + -62.817;
   1:  PR[GP1:91,2] = PR[GP1:90,2] + 0.261;
   1:L PR[91] 10mm/sec CNT100;
   1:  PR[GP1:91,1] = PR[GP1:90,1] + -62.337;
   1:  PR[GP1:91,2] = PR[GP1:90,2] + -4.054;
   1:L PR[91] 10mm/sec CNT100;
   1:  PR[GP1:91,1] = PR[GP1:90,1] + -61.338;
   1:  PR[GP1:91,2] = PR[GP1:90,2] + -9.895;
   1:L PR[91] 10mm/sec CNT100;
   1:  PR[GP1:91,1] = PR[GP1:90,1] + -59.820;
   1:  PR[GP1:91,2] = PR[GP1:90,2] + -14.076;
   1:L PR[91] 10mm/sec CNT100;
   1:  PR[GP1:91,1] = PR[GP1:90,1] + -56.799;
   1:  PR[GP1:91,2] = PR[GP1:90,2] + -19.547;
   1:L PR[91] 10mm/sec CNT100;
   1:  PR[GP1:91,1] = PR[GP1:90,1] + -54.427;
   1:  PR[GP1:91,2] = PR[GP1:90,2] + -23.249;
   1:L PR[91] 10mm/sec CNT100;
   1:  PR[GP1:91,1] = PR[GP1:90,1] + -51.538;
   1:  PR[GP1:91,2] = PR[GP1:90,2] + -26.083;
   1:L PR[91] 10mm/sec CNT100;
   1:  PR[GP1:91,1] = PR[GP1:90,1] + -46.396;
   1:  PR[GP1:91,2] = PR[GP1:90,2] + -30.748;
   1:L PR[91] 10mm/sec CNT100;
   1:  PR[GP1:91,1] = PR[GP1:90,1] + -43.082;
   1:  PR[GP1:91,2] = PR[GP1:90,2] + -32.838;
   1:L PR[91] 10mm/sec CNT100;
   1:  PR[GP1:91,1] = PR[GP1:90,1] + -36.054;
   1:  PR[GP1:91,2] = PR[GP1:90,2] + -35.931;
   1:L PR[91] 10mm/sec CNT100;
   1:  PR[GP1:91,1] = PR[GP1:90,1] + -32.596;
   1:  PR[GP1:91,2] = PR[GP1:90,2] + -37.197;
   1:L PR[91] 10mm/sec CNT100;
   1:  PR[GP1:91,1] = PR[GP1:90,1] + -29.309;
   1:  PR[GP1:91,2] = PR[GP1:90,2] + -37.665;
   1:L PR[91] 10mm/sec CNT100;
   1:  PR[GP1:91,1] = PR[GP1:90,1] + -20.801;
   1:  PR[GP1:91,2] = PR[GP1:90,2] + -38.481;
   1:L PR[91] 10mm/sec CNT100;
   1:  PR[GP1:91,1] = PR[GP1:90,1] + -17.797;
   1:  PR[GP1:91,2] = PR[GP1:90,2] + -38.283;
   1:L PR[91] 10mm/sec CNT100;
   1:  PR[GP1:91,1] = PR[GP1:90,1] + -8.768;
   1:  PR[GP1:91,2] = PR[GP1:90,2] + -36.217;
   1:L PR[91] 10mm/sec CNT100;
   1:  PR[GP1:91,1] = PR[GP1:90,1] + -6.172;
   1:  PR[GP1:91,2] = PR[GP1:90,2] + -35.472;
   1:L PR[91] 10mm/sec CNT100;
   1:  PR[GP1:91,1] = PR[GP1:90,1] + -0.266;
   1:  PR[GP1:91,2] = PR[GP1:90,2] + -32.012;
   1:L PR[91] 10mm/sec CNT100;
   1:  PR[GP1:91,1] = PR[GP1:90,1] + 5.388;
   1:  PR[GP1:91,2] = PR[GP1:90,2] + -35.540;
   1:  PR[GP1:91,3] = PR[GP1:90,3] + 71.675;
   1:L PR[91] 10mm/sec CNT100;
   1:  PR[GP1:91,1] = PR[GP1:90,1] + 7.867;
   1:  PR[GP1:91,2] = PR[GP1:90,2] + -36.252;
   1:L PR[91] 10mm/sec CNT100;
   1:  PR[GP1:91,1] = PR[GP1:90,1] + 17.095;
   1:  PR[GP1:91,2] = PR[GP1:90,2] + -38.363;
   1:L PR[91] 10mm/sec CNT100;
   1:  PR[GP1:91,1] = PR[GP1:90,1] + 19.954;
   1:  PR[GP1:91,2] = PR[GP1:90,2] + -38.553;
   1:L PR[91] 10mm/sec CNT100;
   1:  PR[GP1:91,1] = PR[GP1:90,1] + 23.185;
   1:  PR[GP1:91,2] = PR[GP1:90,2] + -38.107;
   1:L PR[91] 10mm/sec CNT100;
   1:  PR[GP1:91,1] = PR[GP1:90,1] + 31.847;
   1:  PR[GP1:91,2] = PR[GP1:90,2] + -37.265;
   1:L PR[91] 10mm/sec CNT100;
   1:  PR[GP1:91,1] = PR[GP1:90,1] + 35.169;
   1:  PR[GP1:91,2] = PR[GP1:90,2] + -36.053;
   1:L PR[91] 10mm/sec CNT100;
   1:  PR[GP1:91,1] = PR[GP1:90,1] + 42.398;
   1:  PR[GP1:91,2] = PR[GP1:90,2] + -32.874;
   1:L PR[91] 10mm/sec CNT100;
   1:  PR[GP1:91,1] = PR[GP1:90,1] + 45.571;
   1:  PR[GP1:91,2] = PR[GP1:90,2] + -30.883;
   1:L PR[91] 10mm/sec CNT100;
   1:  PR[GP1:91,1] = PR[GP1:90,1] + 48.474;
   1:  PR[GP1:91,2] = PR[GP1:90,2] + -28.054;
   1:L PR[91] 10mm/sec CNT100;
   1:  PR[GP1:91,1] = PR[GP1:90,1] + 53.683;
   1:  PR[GP1:91,2] = PR[GP1:90,2] + -23.316;
   1:L PR[91] 10mm/sec CNT100;
   1:  PR[GP1:91,1] = PR[GP1:90,1] + 55.999;
   1:  PR[GP1:91,2] = PR[GP1:90,2] + -19.723;
   1:L PR[91] 10mm/sec CNT100;
   1:  PR[GP1:91,1] = PR[GP1:90,1] + 59.128;
   1:  PR[GP1:91,2] = PR[GP1:90,2] + -14.067;
   1:L PR[91] 10mm/sec CNT100;
   1:  PR[GP1:91,1] = PR[GP1:90,1] + 60.588;
   1:  PR[GP1:91,2] = PR[GP1:90,2] + -10.098;
   1:L PR[91] 10mm/sec CNT100;
   1:  PR[GP1:91,1] = PR[GP1:90,1] + 61.081;
   1:  PR[GP1:91,2] = PR[GP1:90,2] + -5.758;
   1:L PR[91] 10mm/sec CNT100;
   1:  PR[GP1:91,1] = PR[GP1:90,1] + 62.114;
   1:  PR[GP1:91,2] = PR[GP1:90,2] + 0.296;
   1:L PR[91] 10mm/sec CNT100;
   1:  PR[GP1:91,1] = PR[GP1:90,1] + 61.630;
   1:  PR[GP1:91,2] = PR[GP1:90,2] + 4.576;
   1:L PR[91] 10mm/sec CNT100;
   1:  PR[GP1:91,1] = PR[GP1:90,1] + 60.589;
   1:  PR[GP1:91,2] = PR[GP1:90,2] + 10.653;
   1:L PR[91] 10mm/sec CNT100;
   1:  PR[GP1:91,1] = PR[GP1:90,1] + 59.124;
   1:  PR[GP1:91,2] = PR[GP1:90,2] + 14.637;
   1:L PR[91] 10mm/sec CNT100;
   1:  PR[GP1:91,1] = PR[GP1:90,1] + 55.981;
   1:  PR[GP1:91,2] = PR[GP1:90,2] + 20.303;
   1:L PR[91] 10mm/sec CNT100;
   1:  PR[GP1:91,1] = PR[GP1:90,1] + 53.658;
   1:  PR[GP1:91,2] = PR[GP1:90,2] + 23.906;
   1:L PR[91] 10mm/sec CNT100;
   1:  PR[GP1:91,1] = PR[GP1:90,1] + 50.864;
   1:  PR[GP1:91,2] = PR[GP1:90,2] + 26.643;
   1:L PR[91] 10mm/sec CNT100;
   1:  PR[GP1:91,1] = PR[GP1:90,1] + 45.540;
   1:  PR[GP1:91,2] = PR[GP1:90,2] + 31.461;
   1:L PR[91] 10mm/sec CNT100;
   1:  PR[GP1:91,1] = PR[GP1:90,1] + 42.357;
   1:  PR[GP1:91,2] = PR[GP1:90,2] + 33.459;
   1:L PR[91] 10mm/sec CNT100;
   1:  PR[GP1:91,1] = PR[GP1:90,1] + 35.101;
   1:  PR[GP1:91,2] = PR[GP1:90,2] + 36.629;
   1:L PR[91] 10mm/sec CNT100;
   1:  PR[GP1:91,1] = PR[GP1:90,1] + 31.764;
   1:  PR[GP1:91,2] = PR[GP1:90,2] + 37.846;
   1:L PR[91] 10mm/sec CNT100;
   1:  PR[GP1:91,1] = PR[GP1:90,1] + 28.608;
   1:  PR[GP1:91,2] = PR[GP1:90,2] + 38.294;
   1:L PR[91] 10mm/sec CNT100;
   1:  PR[GP1:91,1] = PR[GP1:90,1] + 19.868;
   1:  PR[GP1:91,2] = PR[GP1:90,2] + 39.106;
   1:L PR[91] 10mm/sec CNT100;
   1:  PR[GP1:91,1] = PR[GP1:90,1] + 16.999;
   1:  PR[GP1:91,2] = PR[GP1:90,2] + 38.915;
   1:L PR[91] 10mm/sec CNT100;
   1:  PR[GP1:91,1] = PR[GP1:90,1] + 7.619;
   1:  PR[GP1:91,2] = PR[GP1:90,2] + 36.700;
   1:L PR[91] 10mm/sec CNT100;
   1:  PR[GP1:91,1] = PR[GP1:90,1] + 5.204;
   1:  PR[GP1:91,2] = PR[GP1:90,2] + 36.006;
   1:L PR[91] 10mm/sec CNT100;
   1:  PR[GP1:91,1] = PR[GP1:90,1] + 2.438;
   1:  PR[GP1:91,2] = PR[GP1:90,2] + 34.532;
   1:L PR[91] 10mm/sec CNT100;
   1:  PR[GP1:91,1] = PR[GP1:90,1] + -0.263;
   1:  PR[GP1:91,2] = PR[GP1:90,2] + 32.335;
   1:L PR[91] 10mm/sec CNT100;
   1:  PR[GP1:91,1] = PR[GP1:90,1] + -2.958;
   1:  PR[GP1:91,2] = PR[GP1:90,2] + 34.526;
   1:L PR[91] 10mm/sec CNT100;
   1:  PR[GP1:91,1] = PR[GP1:90,1] + -5.730;
   1:  PR[GP1:91,2] = PR[GP1:90,2] + 36.007;
   1:L PR[91] 10mm/sec CNT100;
   1:  PR[GP1:91,1] = PR[GP1:90,1] + -8.141;
   1:  PR[GP1:91,2] = PR[GP1:90,2] + 36.700;
   1:L PR[91] 10mm/sec CNT100;
   1:  PR[GP1:91,1] = PR[GP1:90,1] + -17.523;
   1:  PR[GP1:91,2] = PR[GP1:90,2] + 38.915;
   1:L PR[91] 10mm/sec CNT100;
   1:  PR[GP1:91,1] = PR[GP1:90,1] + -20.388;
   1:  PR[GP1:91,2] = PR[GP1:90,2] + 39.104;
   1:L PR[91] 10mm/sec CNT100;
   1:  PR[GP1:91,1] = PR[GP1:90,1] + -23.632;
   1:  PR[GP1:91,2] = PR[GP1:90,2] + 38.655;
   1:L PR[91] 10mm/sec CNT100;
   1:  PR[GP1:91,1] = PR[GP1:90,1] + -32.321;
   1:  PR[GP1:91,2] = PR[GP1:90,2] + 37.838;
   1:L PR[91] 10mm/sec CNT100;
   1:  PR[GP1:91,1] = PR[GP1:90,1] + -35.640;
   1:  PR[GP1:91,2] = PR[GP1:90,2] + 36.623;
   1:L PR[91] 10mm/sec CNT100;
   1:  PR[GP1:91,1] = PR[GP1:90,1] + -42.896;
   1:  PR[GP1:91,2] = PR[GP1:90,2] + 33.451;
   1:L PR[91] 10mm/sec CNT100;
   1:  PR[GP1:91,1] = PR[GP1:90,1] + -46.089;
   1:  PR[GP1:91,2] = PR[GP1:90,2] + 31.437;
   1:L PR[91] 10mm/sec CNT100;
   1:  PR[GP1:91,1] = PR[GP1:90,1] + -48.998;
   1:  PR[GP1:91,2] = PR[GP1:90,2] + 28.597;
   1:L PR[91] 10mm/sec CNT100;
   1:  PR[GP1:91,1] = PR[GP1:90,1] + -54.227;
   1:  PR[GP1:91,2] = PR[GP1:90,2] + 23.863;
   1:L PR[91] 10mm/sec CNT100;
   1:  PR[GP1:91,1] = PR[GP1:90,1] + -56.519;
   1:  PR[GP1:91,2] = PR[GP1:90,2] + 20.286;
   1:L PR[91] 10mm/sec CNT100;
   1:  PR[GP1:91,1] = PR[GP1:90,1] + -59.661;
   1:  PR[GP1:91,2] = PR[GP1:90,2] + 14.610;
   1:L PR[91] 10mm/sec CNT100;
   1:  PR[GP1:91,1] = PR[GP1:90,1] + -61.127;
   1:  PR[GP1:91,2] = PR[GP1:90,2] + 10.571;
   1:L PR[91] 10mm/sec CNT100;
   1:  PR[GP1:91,1] = PR[GP1:90,1] + -61.603;
   1:  PR[GP1:91,2] = PR[GP1:90,2] + 6.323;
   1:L PR[91] 10mm/sec CNT100;
   1:  PR[GP1:91,1] = PR[GP1:90,1] + -62.640;
   1:  PR[GP1:91,2] = PR[GP1:90,2] + 0.261;
   1:L PR[91] 10mm/sec CNT100;
   1:  PR[GP1:91,1] = PR[GP1:90,1] + -62.174;
   1:  PR[GP1:91,2] = PR[GP1:90,2] + -3.926;
   1:L PR[91] 10mm/sec CNT100;
   1:  PR[GP1:91,1] = PR[GP1:90,1] + -61.138;
   1:  PR[GP1:91,2] = PR[GP1:90,2] + -9.984;
   1:L PR[91] 10mm/sec CNT100;
   1:  PR[GP1:91,1] = PR[GP1:90,1] + -59.666;
   1:  PR[GP1:91,2] = PR[GP1:90,2] + -14.039;
   1:L PR[91] 10mm/sec CNT100;
   1:  PR[GP1:91,1] = PR[GP1:90,1] + -56.537;
   1:  PR[GP1:91,2] = PR[GP1:90,2] + -19.705;
   1:L PR[91] 10mm/sec CNT100;
   1:  PR[GP1:91,1] = PR[GP1:90,1] + -54.239;
   1:  PR[GP1:91,2] = PR[GP1:90,2] + -23.292;
   1:L PR[91] 10mm/sec CNT100;
   1:  PR[GP1:91,1] = PR[GP1:90,1] + -51.440;
   1:  PR[GP1:91,2] = PR[GP1:90,2] + -26.037;
   1:L PR[91] 10mm/sec CNT100;
   1:  PR[GP1:91,1] = PR[GP1:90,1] + -46.139;
   1:  PR[GP1:91,2] = PR[GP1:90,2] + -30.847;
   1:L PR[91] 10mm/sec CNT100;
   1:  PR[GP1:91,1] = PR[GP1:90,1] + -42.937;
   1:  PR[GP1:91,2] = PR[GP1:90,2] + -32.866;
   1:L PR[91] 10mm/sec CNT100;
   1:  PR[GP1:91,1] = PR[GP1:90,1] + -35.709;
   1:  PR[GP1:91,2] = PR[GP1:90,2] + -36.047;
   1:L PR[91] 10mm/sec CNT100;
   1:  PR[GP1:91,1] = PR[GP1:90,1] + -32.378;
   1:  PR[GP1:91,2] = PR[GP1:90,2] + -37.267;
   1:L PR[91] 10mm/sec CNT100;
   1:  PR[GP1:91,1] = PR[GP1:90,1] + -29.212;
   1:  PR[GP1:91,2] = PR[GP1:90,2] + -37.718;
   1:L PR[91] 10mm/sec CNT100;
   1:  PR[GP1:91,1] = PR[GP1:90,1] + -20.500;
   1:  PR[GP1:91,2] = PR[GP1:90,2] + -38.553;
   1:L PR[91] 10mm/sec CNT100;
   1:  PR[GP1:91,1] = PR[GP1:90,1] + -17.621;
   1:  PR[GP1:91,2] = PR[GP1:90,2] + -38.363;
   1:L PR[91] 10mm/sec CNT100;
   1:  PR[GP1:91,1] = PR[GP1:90,1] + -8.393;
   1:  PR[GP1:91,2] = PR[GP1:90,2] + -36.252;
   1:L PR[91] 10mm/sec CNT100;
   1:  PR[GP1:91,1] = PR[GP1:90,1] + -5.917;
   1:  PR[GP1:91,2] = PR[GP1:90,2] + -35.541;
   1:L PR[91] 10mm/sec CNT100;
   1:  PR[GP1:91,1] = PR[GP1:90,1] + -0.266;
   1:  PR[GP1:91,2] = PR[GP1:90,2] + -32.230;
   1:L PR[91] 10mm/sec CNT100;
   1:  PR[GP1:91,1] = PR[GP1:90,1] + 5.134;
   1:  PR[GP1:91,2] = PR[GP1:90,2] + -35.609;
   1:  PR[GP1:91,3] = PR[GP1:90,3] + 72.285;
   1:L PR[91] 10mm/sec CNT100;
   1:  PR[GP1:91,1] = PR[GP1:90,1] + 7.492;
   1:  PR[GP1:91,2] = PR[GP1:90,2] + -36.287;
   1:L PR[91] 10mm/sec CNT100;
   1:  PR[GP1:91,1] = PR[GP1:90,1] + 16.919;
   1:  PR[GP1:91,2] = PR[GP1:90,2] + -38.444;
   1:L PR[91] 10mm/sec CNT100;
   1:  PR[GP1:91,1] = PR[GP1:90,1] + 19.654;
   1:  PR[GP1:91,2] = PR[GP1:90,2] + -38.625;
   1:L PR[91] 10mm/sec CNT100;
   1:  PR[GP1:91,1] = PR[GP1:90,1] + 22.749;
   1:  PR[GP1:91,2] = PR[GP1:90,2] + -38.198;
   1:L PR[91] 10mm/sec CNT100;
   1:  PR[GP1:91,1] = PR[GP1:90,1] + 31.629;
   1:  PR[GP1:91,2] = PR[GP1:90,2] + -37.335;
   1:L PR[91] 10mm/sec CNT100;
   1:  PR[GP1:91,1] = PR[GP1:90,1] + 34.825;
   1:  PR[GP1:91,2] = PR[GP1:90,2] + -36.169;
   1:L PR[91] 10mm/sec CNT100;
   1:  PR[GP1:91,1] = PR[GP1:90,1] + 42.252;
   1:  PR[GP1:91,2] = PR[GP1:90,2] + -32.902;
   1:L PR[91] 10mm/sec CNT100;
   1:  PR[GP1:91,1] = PR[GP1:90,1] + 45.316;
   1:  PR[GP1:91,2] = PR[GP1:90,2] + -30.980;
   1:L PR[91] 10mm/sec CNT100;
   1:  PR[GP1:91,1] = PR[GP1:90,1] + 48.119;
   1:  PR[GP1:91,2] = PR[GP1:90,2] + -28.248;
   1:L PR[91] 10mm/sec CNT100;
   1:  PR[GP1:91,1] = PR[GP1:90,1] + 53.496;
   1:  PR[GP1:91,2] = PR[GP1:90,2] + -23.357;
   1:L PR[91] 10mm/sec CNT100;
   1:  PR[GP1:91,1] = PR[GP1:90,1] + 55.737;
   1:  PR[GP1:91,2] = PR[GP1:90,2] + -19.880;
   1:L PR[91] 10mm/sec CNT100;
   1:  PR[GP1:91,1] = PR[GP1:90,1] + 58.974;
   1:  PR[GP1:91,2] = PR[GP1:90,2] + -14.030;
   1:L PR[91] 10mm/sec CNT100;
   1:  PR[GP1:91,1] = PR[GP1:90,1] + 60.388;
   1:  PR[GP1:91,2] = PR[GP1:90,2] + -10.185;
   1:L PR[91] 10mm/sec CNT100;
   1:  PR[GP1:91,1] = PR[GP1:90,1] + 60.866;
   1:  PR[GP1:91,2] = PR[GP1:90,2] + -5.978;
   1:L PR[91] 10mm/sec CNT100;
   1:  PR[GP1:91,1] = PR[GP1:90,1] + 61.937;
   1:  PR[GP1:91,2] = PR[GP1:90,2] + 0.296;
   1:L PR[91] 10mm/sec CNT100;
   1:  PR[GP1:91,1] = PR[GP1:90,1] + 61.467;
   1:  PR[GP1:91,2] = PR[GP1:90,2] + 4.445;
   1:L PR[91] 10mm/sec CNT100;
   1:  PR[GP1:91,1] = PR[GP1:90,1] + 60.390;
   1:  PR[GP1:91,2] = PR[GP1:90,2] + 10.740;
   1:L PR[91] 10mm/sec CNT100;
   1:  PR[GP1:91,1] = PR[GP1:90,1] + 58.970;
   1:  PR[GP1:91,2] = PR[GP1:90,2] + 14.601;
   1:L PR[91] 10mm/sec CNT100;
   1:  PR[GP1:91,1] = PR[GP1:90,1] + 55.719;
   1:  PR[GP1:91,2] = PR[GP1:90,2] + 20.462;
   1:L PR[91] 10mm/sec CNT100;
   1:  PR[GP1:91,1] = PR[GP1:90,1] + 53.471;
   1:  PR[GP1:91,2] = PR[GP1:90,2] + 23.949;
   1:L PR[91] 10mm/sec CNT100;
   1:  PR[GP1:91,1] = PR[GP1:90,1] + 50.766;
   1:  PR[GP1:91,2] = PR[GP1:90,2] + 26.597;
   1:L PR[91] 10mm/sec CNT100;
   1:  PR[GP1:91,1] = PR[GP1:90,1] + 45.283;
   1:  PR[GP1:91,2] = PR[GP1:90,2] + 31.560;
   1:L PR[91] 10mm/sec CNT100;
   1:  PR[GP1:91,1] = PR[GP1:90,1] + 42.210;
   1:  PR[GP1:91,2] = PR[GP1:90,2] + 33.488;
   1:L PR[91] 10mm/sec CNT100;
   1:  PR[GP1:91,1] = PR[GP1:90,1] + 34.755;
   1:  PR[GP1:91,2] = PR[GP1:90,2] + 36.745;
   1:L PR[91] 10mm/sec CNT100;
   1:  PR[GP1:91,1] = PR[GP1:90,1] + 31.545;
   1:  PR[GP1:91,2] = PR[GP1:90,2] + 37.916;
   1:L PR[91] 10mm/sec CNT100;
   1:  PR[GP1:91,1] = PR[GP1:90,1] + 28.509;
   1:  PR[GP1:91,2] = PR[GP1:90,2] + 38.347;
   1:L PR[91] 10mm/sec CNT100;
   1:  PR[GP1:91,1] = PR[GP1:90,1] + 19.566;
   1:  PR[GP1:91,2] = PR[GP1:90,2] + 39.178;
   1:L PR[91] 10mm/sec CNT100;
   1:  PR[GP1:91,1] = PR[GP1:90,1] + 16.820;
   1:  PR[GP1:91,2] = PR[GP1:90,2] + 38.995;
   1:L PR[91] 10mm/sec CNT100;
   1:  PR[GP1:91,1] = PR[GP1:90,1] + 7.238;
   1:  PR[GP1:91,2] = PR[GP1:90,2] + 36.732;
   1:L PR[91] 10mm/sec CNT100;
   1:  PR[GP1:91,1] = PR[GP1:90,1] + 4.946;
   1:  PR[GP1:91,2] = PR[GP1:90,2] + 36.073;
   1:L PR[91] 10mm/sec CNT100;
   1:  PR[GP1:91,1] = PR[GP1:90,1] + 2.265;
   1:  PR[GP1:91,2] = PR[GP1:90,2] + 34.646;
   1:L PR[91] 10mm/sec CNT100;
   1:  PR[GP1:91,1] = PR[GP1:90,1] + -0.263;
   1:  PR[GP1:91,2] = PR[GP1:90,2] + 32.590;
   1:L PR[91] 10mm/sec CNT100;
   1:  PR[GP1:91,1] = PR[GP1:90,1] + -2.786;
   1:  PR[GP1:91,2] = PR[GP1:90,2] + 34.641;
   1:L PR[91] 10mm/sec CNT100;
   1:  PR[GP1:91,1] = PR[GP1:90,1] + -5.471;
   1:  PR[GP1:91,2] = PR[GP1:90,2] + 36.075;
   1:L PR[91] 10mm/sec CNT100;
   1:  PR[GP1:91,1] = PR[GP1:90,1] + -7.760;
   1:  PR[GP1:91,2] = PR[GP1:90,2] + 36.733;
   1:L PR[91] 10mm/sec CNT100;
   1:  PR[GP1:91,1] = PR[GP1:90,1] + -17.344;
   1:  PR[GP1:91,2] = PR[GP1:90,2] + 38.995;
   1:L PR[91] 10mm/sec CNT100;
   1:  PR[GP1:91,1] = PR[GP1:90,1] + -20.086;
   1:  PR[GP1:91,2] = PR[GP1:90,2] + 39.176;
   1:L PR[91] 10mm/sec CNT100;
   1:  PR[GP1:91,1] = PR[GP1:90,1] + -23.192;
   1:  PR[GP1:91,2] = PR[GP1:90,2] + 38.746;
   1:L PR[91] 10mm/sec CNT100;
   1:  PR[GP1:91,1] = PR[GP1:90,1] + -32.102;
   1:  PR[GP1:91,2] = PR[GP1:90,2] + 37.909;
   1:L PR[91] 10mm/sec CNT100;
   1:  PR[GP1:91,1] = PR[GP1:90,1] + -35.294;
   1:  PR[GP1:91,2] = PR[GP1:90,2] + 36.740;
   1:L PR[91] 10mm/sec CNT100;
   1:  PR[GP1:91,1] = PR[GP1:90,1] + -42.749;
   1:  PR[GP1:91,2] = PR[GP1:90,2] + 33.480;
   1:L PR[91] 10mm/sec CNT100;
   1:  PR[GP1:91,1] = PR[GP1:90,1] + -45.831;
   1:  PR[GP1:91,2] = PR[GP1:90,2] + 31.537;
   1:L PR[91] 10mm/sec CNT100;
   1:  PR[GP1:91,1] = PR[GP1:90,1] + -48.641;
   1:  PR[GP1:91,2] = PR[GP1:90,2] + 28.794;
   1:L PR[91] 10mm/sec CNT100;
   1:  PR[GP1:91,1] = PR[GP1:90,1] + -54.039;
   1:  PR[GP1:91,2] = PR[GP1:90,2] + 23.906;
   1:L PR[91] 10mm/sec CNT100;
   1:  PR[GP1:91,1] = PR[GP1:90,1] + -56.256;
   1:  PR[GP1:91,2] = PR[GP1:90,2] + 20.445;
   1:L PR[91] 10mm/sec CNT100;
   1:  PR[GP1:91,1] = PR[GP1:90,1] + -59.507;
   1:  PR[GP1:91,2] = PR[GP1:90,2] + 14.574;
   1:L PR[91] 10mm/sec CNT100;
   1:  PR[GP1:91,1] = PR[GP1:90,1] + -60.927;
   1:  PR[GP1:91,2] = PR[GP1:90,2] + 10.661;
   1:L PR[91] 10mm/sec CNT100;
   1:  PR[GP1:91,1] = PR[GP1:90,1] + -61.388;
   1:  PR[GP1:91,2] = PR[GP1:90,2] + 6.543;
   1:L PR[91] 10mm/sec CNT100;
   1:  PR[GP1:91,1] = PR[GP1:90,1] + -62.463;
   1:  PR[GP1:91,2] = PR[GP1:90,2] + 0.261;
   1:L PR[91] 10mm/sec CNT100;
   1:  PR[GP1:91,1] = PR[GP1:90,1] + -62.011;
   1:  PR[GP1:91,2] = PR[GP1:90,2] + -3.798;
   1:L PR[91] 10mm/sec CNT100;
   1:  PR[GP1:91,1] = PR[GP1:90,1] + -60.938;
   1:  PR[GP1:91,2] = PR[GP1:90,2] + -10.073;
   1:L PR[91] 10mm/sec CNT100;
   1:  PR[GP1:91,1] = PR[GP1:90,1] + -59.511;
   1:  PR[GP1:91,2] = PR[GP1:90,2] + -14.003;
   1:L PR[91] 10mm/sec CNT100;
   1:  PR[GP1:91,1] = PR[GP1:90,1] + -56.275;
   1:  PR[GP1:91,2] = PR[GP1:90,2] + -19.864;
   1:L PR[91] 10mm/sec CNT100;
   1:  PR[GP1:91,1] = PR[GP1:90,1] + -54.051;
   1:  PR[GP1:91,2] = PR[GP1:90,2] + -23.335;
   1:L PR[91] 10mm/sec CNT100;
   1:  PR[GP1:91,1] = PR[GP1:90,1] + -51.343;
   1:  PR[GP1:91,2] = PR[GP1:90,2] + -25.992;
   1:L PR[91] 10mm/sec CNT100;
   1:  PR[GP1:91,1] = PR[GP1:90,1] + -45.882;
   1:  PR[GP1:91,2] = PR[GP1:90,2] + -30.945;
   1:L PR[91] 10mm/sec CNT100;
   1:  PR[GP1:91,1] = PR[GP1:90,1] + -42.791;
   1:  PR[GP1:91,2] = PR[GP1:90,2] + -32.895;
   1:L PR[91] 10mm/sec CNT100;
   1:  PR[GP1:91,1] = PR[GP1:90,1] + -35.365;
   1:  PR[GP1:91,2] = PR[GP1:90,2] + -36.163;
   1:L PR[91] 10mm/sec CNT100;
   1:  PR[GP1:91,1] = PR[GP1:90,1] + -32.160;
   1:  PR[GP1:91,2] = PR[GP1:90,2] + -37.337;
   1:L PR[91] 10mm/sec CNT100;
   1:  PR[GP1:91,1] = PR[GP1:90,1] + -29.114;
   1:  PR[GP1:91,2] = PR[GP1:90,2] + -37.770;
   1:L PR[91] 10mm/sec CNT100;
   1:  PR[GP1:91,1] = PR[GP1:90,1] + -20.200;
   1:  PR[GP1:91,2] = PR[GP1:90,2] + -38.625;
   1:L PR[91] 10mm/sec CNT100;
   1:  PR[GP1:91,1] = PR[GP1:90,1] + -17.444;
   1:  PR[GP1:91,2] = PR[GP1:90,2] + -38.444;
   1:L PR[91] 10mm/sec CNT100;
   1:  PR[GP1:91,1] = PR[GP1:90,1] + -8.017;
   1:  PR[GP1:91,2] = PR[GP1:90,2] + -36.287;
   1:L PR[91] 10mm/sec CNT100;
   1:  PR[GP1:91,1] = PR[GP1:90,1] + -5.663;
   1:  PR[GP1:91,2] = PR[GP1:90,2] + -35.611;
   1:L PR[91] 10mm/sec CNT100;
   1:  PR[GP1:91,1] = PR[GP1:90,1] + -0.266;
   1:  PR[GP1:91,2] = PR[GP1:90,2] + -32.449;
   1:L PR[91] 10mm/sec CNT100;
   1:  PR[GP1:91,1] = PR[GP1:90,1] + 4.879;
   1:  PR[GP1:91,2] = PR[GP1:90,2] + -35.679;
   1:  PR[GP1:91,3] = PR[GP1:90,3] + 72.895;
   1:L PR[91] 10mm/sec CNT100;
   1:  PR[GP1:91,1] = PR[GP1:90,1] + 7.117;
   1:  PR[GP1:91,2] = PR[GP1:90,2] + -36.321;
   1:L PR[91] 10mm/sec CNT100;
   1:  PR[GP1:91,1] = PR[GP1:90,1] + 16.742;
   1:  PR[GP1:91,2] = PR[GP1:90,2] + -38.524;
   1:L PR[91] 10mm/sec CNT100;
   1:  PR[GP1:91,1] = PR[GP1:90,1] + 19.354;
   1:  PR[GP1:91,2] = PR[GP1:90,2] + -38.697;
   1:L PR[91] 10mm/sec CNT100;
   1:  PR[GP1:91,1] = PR[GP1:90,1] + 22.313;
   1:  PR[GP1:91,2] = PR[GP1:90,2] + -38.289;
   1:L PR[91] 10mm/sec CNT100;
   1:  PR[GP1:91,1] = PR[GP1:90,1] + 31.412;
   1:  PR[GP1:91,2] = PR[GP1:90,2] + -37.404;
   1:L PR[91] 10mm/sec CNT100;
   1:  PR[GP1:91,1] = PR[GP1:90,1] + 34.481;
   1:  PR[GP1:91,2] = PR[GP1:90,2] + -36.284;
   1:L PR[91] 10mm/sec CNT100;
   1:  PR[GP1:91,1] = PR[GP1:90,1] + 42.107;
   1:  PR[GP1:91,2] = PR[GP1:90,2] + -32.931;
   1:L PR[91] 10mm/sec CNT100;
   1:  PR[GP1:91,1] = PR[GP1:90,1] + 45.060;
   1:  PR[GP1:91,2] = PR[GP1:90,2] + -31.078;
   1:L PR[91] 10mm/sec CNT100;
   1:  PR[GP1:91,1] = PR[GP1:90,1] + 47.764;
   1:  PR[GP1:91,2] = PR[GP1:90,2] + -28.443;
   1:L PR[91] 10mm/sec CNT100;
   1:  PR[GP1:91,1] = PR[GP1:90,1] + 53.309;
   1:  PR[GP1:91,2] = PR[GP1:90,2] + -23.399;
   1:L PR[91] 10mm/sec CNT100;
   1:  PR[GP1:91,1] = PR[GP1:90,1] + 55.476;
   1:  PR[GP1:91,2] = PR[GP1:90,2] + -20.038;
   1:L PR[91] 10mm/sec CNT100;
   1:  PR[GP1:91,1] = PR[GP1:90,1] + 58.820;
   1:  PR[GP1:91,2] = PR[GP1:90,2] + -13.993;
   1:L PR[91] 10mm/sec CNT100;
   1:  PR[GP1:91,1] = PR[GP1:90,1] + 60.189;
   1:  PR[GP1:91,2] = PR[GP1:90,2] + -10.271;
   1:L PR[91] 10mm/sec CNT100;
   1:  PR[GP1:91,1] = PR[GP1:90,1] + 60.652;
   1:  PR[GP1:91,2] = PR[GP1:90,2] + -6.198;
   1:L PR[91] 10mm/sec CNT100;
   1:  PR[GP1:91,1] = PR[GP1:90,1] + 61.759;
   1:  PR[GP1:91,2] = PR[GP1:90,2] + 0.296;
   1:L PR[91] 10mm/sec CNT100;
   1:  PR[GP1:91,1] = PR[GP1:90,1] + 61.305;
   1:  PR[GP1:91,2] = PR[GP1:90,2] + 4.314;
   1:L PR[91] 10mm/sec CNT100;
   1:  PR[GP1:91,1] = PR[GP1:90,1] + 60.190;
   1:  PR[GP1:91,2] = PR[GP1:90,2] + 10.827;
   1:L PR[91] 10mm/sec CNT100;
   1:  PR[GP1:91,1] = PR[GP1:90,1] + 58.815;
   1:  PR[GP1:91,2] = PR[GP1:90,2] + 14.564;
   1:L PR[91] 10mm/sec CNT100;
   1:  PR[GP1:91,1] = PR[GP1:90,1] + 55.457;
   1:  PR[GP1:91,2] = PR[GP1:90,2] + 20.620;
   1:L PR[91] 10mm/sec CNT100;
   1:  PR[GP1:91,1] = PR[GP1:90,1] + 53.283;
   1:  PR[GP1:91,2] = PR[GP1:90,2] + 23.991;
   1:L PR[91] 10mm/sec CNT100;
   1:  PR[GP1:91,1] = PR[GP1:90,1] + 50.669;
   1:  PR[GP1:91,2] = PR[GP1:90,2] + 26.551;
   1:L PR[91] 10mm/sec CNT100;
   1:  PR[GP1:91,1] = PR[GP1:90,1] + 45.026;
   1:  PR[GP1:91,2] = PR[GP1:90,2] + 31.658;
   1:L PR[91] 10mm/sec CNT100;
   1:  PR[GP1:91,1] = PR[GP1:90,1] + 42.064;
   1:  PR[GP1:91,2] = PR[GP1:90,2] + 33.517;
   1:L PR[91] 10mm/sec CNT100;
   1:  PR[GP1:91,1] = PR[GP1:90,1] + 34.409;
   1:  PR[GP1:91,2] = PR[GP1:90,2] + 36.861;
   1:L PR[91] 10mm/sec CNT100;
   1:  PR[GP1:91,1] = PR[GP1:90,1] + 31.326;
   1:  PR[GP1:91,2] = PR[GP1:90,2] + 37.986;
   1:L PR[91] 10mm/sec CNT100;
   1:  PR[GP1:91,1] = PR[GP1:90,1] + 28.409;
   1:  PR[GP1:91,2] = PR[GP1:90,2] + 38.400;
   1:L PR[91] 10mm/sec CNT100;
   1:  PR[GP1:91,1] = PR[GP1:90,1] + 19.264;
   1:  PR[GP1:91,2] = PR[GP1:90,2] + 39.250;
   1:L PR[91] 10mm/sec CNT100;
   1:  PR[GP1:91,1] = PR[GP1:90,1] + 16.641;
   1:  PR[GP1:91,2] = PR[GP1:90,2] + 39.075;
   1:L PR[91] 10mm/sec CNT100;
   1:  PR[GP1:91,1] = PR[GP1:90,1] + 6.858;
   1:  PR[GP1:91,2] = PR[GP1:90,2] + 36.765;
   1:L PR[91] 10mm/sec CNT100;
   1:  PR[GP1:91,1] = PR[GP1:90,1] + 4.688;
   1:  PR[GP1:91,2] = PR[GP1:90,2] + 36.141;
   1:L PR[91] 10mm/sec CNT100;
   1:  PR[GP1:91,1] = PR[GP1:90,1] + 2.092;
   1:  PR[GP1:91,2] = PR[GP1:90,2] + 34.760;
   1:L PR[91] 10mm/sec CNT100;
   1:  PR[GP1:91,1] = PR[GP1:90,1] + -0.263;
   1:  PR[GP1:91,2] = PR[GP1:90,2] + 32.845;
   1:L PR[91] 10mm/sec CNT100;
   1:  PR[GP1:91,1] = PR[GP1:90,1] + -2.613;
   1:  PR[GP1:91,2] = PR[GP1:90,2] + 34.755;
   1:L PR[91] 10mm/sec CNT100;
   1:  PR[GP1:91,1] = PR[GP1:90,1] + -5.213;
   1:  PR[GP1:91,2] = PR[GP1:90,2] + 36.142;
   1:L PR[91] 10mm/sec CNT100;
   1:  PR[GP1:91,1] = PR[GP1:90,1] + -7.380;
   1:  PR[GP1:91,2] = PR[GP1:90,2] + 36.765;
   1:L PR[91] 10mm/sec CNT100;
   1:  PR[GP1:91,1] = PR[GP1:90,1] + -17.166;
   1:  PR[GP1:91,2] = PR[GP1:90,2] + 39.075;
   1:L PR[91] 10mm/sec CNT100;
   1:  PR[GP1:91,1] = PR[GP1:90,1] + -19.783;
   1:  PR[GP1:91,2] = PR[GP1:90,2] + 39.248;
   1:L PR[91] 10mm/sec CNT100;
   1:  PR[GP1:91,1] = PR[GP1:90,1] + -22.753;
   1:  PR[GP1:91,2] = PR[GP1:90,2] + 38.837;
   1:L PR[91] 10mm/sec CNT100;
   1:  PR[GP1:91,1] = PR[GP1:90,1] + -31.882;
   1:  PR[GP1:91,2] = PR[GP1:90,2] + 37.979;
   1:L PR[91] 10mm/sec CNT100;
   1:  PR[GP1:91,1] = PR[GP1:90,1] + -34.947;
   1:  PR[GP1:91,2] = PR[GP1:90,2] + 36.856;
   1:L PR[91] 10mm/sec CNT100;
   1:  PR[GP1:91,1] = PR[GP1:90,1] + -42.602;
   1:  PR[GP1:91,2] = PR[GP1:90,2] + 33.509;
   1:L PR[91] 10mm/sec CNT100;
   1:  PR[GP1:91,1] = PR[GP1:90,1] + -45.573;
   1:  PR[GP1:91,2] = PR[GP1:90,2] + 31.636;
   1:L PR[91] 10mm/sec CNT100;
   1:  PR[GP1:91,1] = PR[GP1:90,1] + -48.283;
   1:  PR[GP1:91,2] = PR[GP1:90,2] + 28.990;
   1:L PR[91] 10mm/sec CNT100;
   1:  PR[GP1:91,1] = PR[GP1:90,1] + -53.850;
   1:  PR[GP1:91,2] = PR[GP1:90,2] + 23.950;
   1:L PR[91] 10mm/sec CNT100;
   1:  PR[GP1:91,1] = PR[GP1:90,1] + -55.994;
   1:  PR[GP1:91,2] = PR[GP1:90,2] + 20.604;
   1:L PR[91] 10mm/sec CNT100;
   1:  PR[GP1:91,1] = PR[GP1:90,1] + -59.352;
   1:  PR[GP1:91,2] = PR[GP1:90,2] + 14.538;
   1:L PR[91] 10mm/sec CNT100;
   1:  PR[GP1:91,1] = PR[GP1:90,1] + -60.727;
   1:  PR[GP1:91,2] = PR[GP1:90,2] + 10.751;
   1:L PR[91] 10mm/sec CNT100;
   1:  PR[GP1:91,1] = PR[GP1:90,1] + -61.173;
   1:  PR[GP1:91,2] = PR[GP1:90,2] + 6.763;
   1:L PR[91] 10mm/sec CNT100;
   1:  PR[GP1:91,1] = PR[GP1:90,1] + -62.286;
   1:  PR[GP1:91,2] = PR[GP1:90,2] + 0.261;
   1:L PR[91] 10mm/sec CNT100;
   1:  PR[GP1:91,1] = PR[GP1:90,1] + -61.848;
   1:  PR[GP1:91,2] = PR[GP1:90,2] + -3.670;
   1:L PR[91] 10mm/sec CNT100;
   1:  PR[GP1:91,1] = PR[GP1:90,1] + -60.737;
   1:  PR[GP1:91,2] = PR[GP1:90,2] + -10.163;
   1:L PR[91] 10mm/sec CNT100;
   1:  PR[GP1:91,1] = PR[GP1:90,1] + -59.357;
   1:  PR[GP1:91,2] = PR[GP1:90,2] + -13.967;
   1:L PR[91] 10mm/sec CNT100;
   1:  PR[GP1:91,1] = PR[GP1:90,1] + -56.013;
   1:  PR[GP1:91,2] = PR[GP1:90,2] + -20.022;
   1:L PR[91] 10mm/sec CNT100;
   1:  PR[GP1:91,1] = PR[GP1:90,1] + -53.863;
   1:  PR[GP1:91,2] = PR[GP1:90,2] + -23.377;
   1:L PR[91] 10mm/sec CNT100;
   1:  PR[GP1:91,1] = PR[GP1:90,1] + -51.245;
   1:  PR[GP1:91,2] = PR[GP1:90,2] + -25.946;
   1:L PR[91] 10mm/sec CNT100;
   1:  PR[GP1:91,1] = PR[GP1:90,1] + -45.626;
   1:  PR[GP1:91,2] = PR[GP1:90,2] + -31.044;
   1:L PR[91] 10mm/sec CNT100;
   1:  PR[GP1:91,1] = PR[GP1:90,1] + -42.645;
   1:  PR[GP1:91,2] = PR[GP1:90,2] + -32.923;
   1:L PR[91] 10mm/sec CNT100;
   1:  PR[GP1:91,1] = PR[GP1:90,1] + -35.020;
   1:  PR[GP1:91,2] = PR[GP1:90,2] + -36.279;
   1:L PR[91] 10mm/sec CNT100;
   1:  PR[GP1:91,1] = PR[GP1:90,1] + -31.942;
   1:  PR[GP1:91,2] = PR[GP1:90,2] + -37.406;
   1:L PR[91] 10mm/sec CNT100;
   1:  PR[GP1:91,1] = PR[GP1:90,1] + -29.016;
   1:  PR[GP1:91,2] = PR[GP1:90,2] + -37.823;
   1:L PR[91] 10mm/sec CNT100;
   1:  PR[GP1:91,1] = PR[GP1:90,1] + -19.900;
   1:  PR[GP1:91,2] = PR[GP1:90,2] + -38.697;
   1:L PR[91] 10mm/sec CNT100;
   1:  PR[GP1:91,1] = PR[GP1:90,1] + -17.267;
   1:  PR[GP1:91,2] = PR[GP1:90,2] + -38.524;
   1:L PR[91] 10mm/sec CNT100;
   1:  PR[GP1:91,1] = PR[GP1:90,1] + -7.642;
   1:  PR[GP1:91,2] = PR[GP1:90,2] + -36.322;
   1:L PR[91] 10mm/sec CNT100;
   1:  PR[GP1:91,1] = PR[GP1:90,1] + -5.408;
   1:  PR[GP1:91,2] = PR[GP1:90,2] + -35.680;
   1:L PR[91] 10mm/sec CNT100;
   1:  PR[GP1:91,1] = PR[GP1:90,1] + -0.266;
   1:  PR[GP1:91,2] = PR[GP1:90,2] + -32.668;
   1:L PR[91] 10mm/sec CNT100;
   1:  PR[GP1:91,1] = PR[GP1:90,1] + 4.624;
   1:  PR[GP1:91,2] = PR[GP1:90,2] + -35.748;
   1:  PR[GP1:91,3] = PR[GP1:90,3] + 73.505;
   1:L PR[91] 10mm/sec CNT100;
   1:  PR[GP1:91,1] = PR[GP1:90,1] + 6.741;
   1:  PR[GP1:91,2] = PR[GP1:90,2] + -36.356;
   1:L PR[91] 10mm/sec CNT100;
   1:  PR[GP1:91,1] = PR[GP1:90,1] + 16.565;
   1:  PR[GP1:91,2] = PR[GP1:90,2] + -38.604;
   1:L PR[91] 10mm/sec CNT100;
   1:  PR[GP1:91,1] = PR[GP1:90,1] + 19.054;
   1:  PR[GP1:91,2] = PR[GP1:90,2] + -38.769;
   1:L PR[91] 10mm/sec CNT100;
   1:  PR[GP1:91,1] = PR[GP1:90,1] + 21.877;
   1:  PR[GP1:91,2] = PR[GP1:90,2] + -38.380;
   1:L PR[91] 10mm/sec CNT100;
   1:  PR[GP1:91,1] = PR[GP1:90,1] + 31.194;
   1:  PR[GP1:91,2] = PR[GP1:90,2] + -37.474;
   1:L PR[91] 10mm/sec CNT100;
   1:  PR[GP1:91,1] = PR[GP1:90,1] + 34.137;
   1:  PR[GP1:91,2] = PR[GP1:90,2] + -36.400;
   1:L PR[91] 10mm/sec CNT100;
   1:  PR[GP1:91,1] = PR[GP1:90,1] + 41.962;
   1:  PR[GP1:91,2] = PR[GP1:90,2] + -32.959;
   1:L PR[91] 10mm/sec CNT100;
   1:  PR[GP1:91,1] = PR[GP1:90,1] + 44.804;
   1:  PR[GP1:91,2] = PR[GP1:90,2] + -31.176;
   1:L PR[91] 10mm/sec CNT100;
   1:  PR[GP1:91,1] = PR[GP1:90,1] + 47.409;
   1:  PR[GP1:91,2] = PR[GP1:90,2] + -28.637;
   1:L PR[91] 10mm/sec CNT100;
   1:  PR[GP1:91,1] = PR[GP1:90,1] + 53.122;
   1:  PR[GP1:91,2] = PR[GP1:90,2] + -23.440;
   1:L PR[91] 10mm/sec CNT100;
   1:  PR[GP1:91,1] = PR[GP1:90,1] + 55.214;
   1:  PR[GP1:91,2] = PR[GP1:90,2] + -20.196;
   1:L PR[91] 10mm/sec CNT100;
   1:  PR[GP1:91,1] = PR[GP1:90,1] + 58.666;
   1:  PR[GP1:91,2] = PR[GP1:90,2] + -13.956;
   1:L PR[91] 10mm/sec CNT100;
   1:  PR[GP1:91,1] = PR[GP1:90,1] + 59.989;
   1:  PR[GP1:91,2] = PR[GP1:90,2] + -10.358;
   1:L PR[91] 10mm/sec CNT100;
   1:  PR[GP1:91,1] = PR[GP1:90,1] + 60.437;
   1:  PR[GP1:91,2] = PR[GP1:90,2] + -6.418;
   1:L PR[91] 10mm/sec CNT100;
   1:  PR[GP1:91,1] = PR[GP1:90,1] + 61.582;
   1:  PR[GP1:91,2] = PR[GP1:90,2] + 0.296;
   1:L PR[91] 10mm/sec CNT100;
   1:  PR[GP1:91,1] = PR[GP1:90,1] + 61.143;
   1:  PR[GP1:91,2] = PR[GP1:90,2] + 4.184;
   1:L PR[91] 10mm/sec CNT100;
   1:  PR[GP1:91,1] = PR[GP1:90,1] + 59.990;
   1:  PR[GP1:91,2] = PR[GP1:90,2] + 10.914;
   1:L PR[91] 10mm/sec CNT100;
   1:  PR[GP1:91,1] = PR[GP1:90,1] + 58.661;
   1:  PR[GP1:91,2] = PR[GP1:90,2] + 14.528;
   1:L PR[91] 10mm/sec CNT100;
   1:  PR[GP1:91,1] = PR[GP1:90,1] + 55.194;
   1:  PR[GP1:91,2] = PR[GP1:90,2] + 20.779;
   1:L PR[91] 10mm/sec CNT100;
   1:  PR[GP1:91,1] = PR[GP1:90,1] + 53.096;
   1:  PR[GP1:91,2] = PR[GP1:90,2] + 24.033;
   1:L PR[91] 10mm/sec CNT100;
   1:  PR[GP1:91,1] = PR[GP1:90,1] + 50.572;
   1:  PR[GP1:91,2] = PR[GP1:90,2] + 26.505;
   1:L PR[91] 10mm/sec CNT100;
   1:  PR[GP1:91,1] = PR[GP1:90,1] + 44.769;
   1:  PR[GP1:91,2] = PR[GP1:90,2] + 31.756;
   1:L PR[91] 10mm/sec CNT100;
   1:  PR[GP1:91,1] = PR[GP1:90,1] + 41.918;
   1:  PR[GP1:91,2] = PR[GP1:90,2] + 33.546;
   1:L PR[91] 10mm/sec CNT100;
   1:  PR[GP1:91,1] = PR[GP1:90,1] + 34.063;
   1:  PR[GP1:91,2] = PR[GP1:90,2] + 36.978;
   1:L PR[91] 10mm/sec CNT100;
   1:  PR[GP1:91,1] = PR[GP1:90,1] + 31.107;
   1:  PR[GP1:91,2] = PR[GP1:90,2] + 38.056;
   1:L PR[91] 10mm/sec CNT100;
   1:  PR[GP1:91,1] = PR[GP1:90,1] + 28.310;
   1:  PR[GP1:91,2] = PR[GP1:90,2] + 38.453;
   1:L PR[91] 10mm/sec CNT100;
   1:  PR[GP1:91,1] = PR[GP1:90,1] + 18.962;
   1:  PR[GP1:91,2] = PR[GP1:90,2] + 39.322;
   1:L PR[91] 10mm/sec CNT100;
   1:  PR[GP1:91,1] = PR[GP1:90,1] + 16.462;
   1:  PR[GP1:91,2] = PR[GP1:90,2] + 39.155;
   1:L PR[91] 10mm/sec CNT100;
   1:  PR[GP1:91,1] = PR[GP1:90,1] + 6.477;
   1:  PR[GP1:91,2] = PR[GP1:90,2] + 36.797;
   1:L PR[91] 10mm/sec CNT100;
   1:  PR[GP1:91,1] = PR[GP1:90,1] + 4.430;
   1:  PR[GP1:91,2] = PR[GP1:90,2] + 36.209;
   1:L PR[91] 10mm/sec CNT100;
   1:  PR[GP1:91,1] = PR[GP1:90,1] + 1.919;
   1:  PR[GP1:91,2] = PR[GP1:90,2] + 34.874;
   1:L PR[91] 10mm/sec CNT100;
   1:  PR[GP1:91,1] = PR[GP1:90,1] + -0.263;
   1:  PR[GP1:91,2] = PR[GP1:90,2] + 33.099;
   1:L PR[91] 10mm/sec CNT100;
   1:  PR[GP1:91,1] = PR[GP1:90,1] + -2.441;
   1:  PR[GP1:91,2] = PR[GP1:90,2] + 34.870;
   1:L PR[91] 10mm/sec CNT100;
   1:  PR[GP1:91,1] = PR[GP1:90,1] + -4.955;
   1:  PR[GP1:91,2] = PR[GP1:90,2] + 36.210;
   1:L PR[91] 10mm/sec CNT100;
   1:  PR[GP1:91,1] = PR[GP1:90,1] + -6.999;
   1:  PR[GP1:91,2] = PR[GP1:90,2] + 36.797;
   1:L PR[91] 10mm/sec CNT100;
   1:  PR[GP1:91,1] = PR[GP1:90,1] + -16.987;
   1:  PR[GP1:91,2] = PR[GP1:90,2] + 39.155;
   1:L PR[91] 10mm/sec CNT100;
   1:  PR[GP1:91,1] = PR[GP1:90,1] + -19.481;
   1:  PR[GP1:91,2] = PR[GP1:90,2] + 39.320;
   1:L PR[91] 10mm/sec CNT100;
   1:  PR[GP1:91,1] = PR[GP1:90,1] + -22.314;
   1:  PR[GP1:91,2] = PR[GP1:90,2] + 38.928;
   1:L PR[91] 10mm/sec CNT100;
   1:  PR[GP1:91,1] = PR[GP1:90,1] + -31.662;
   1:  PR[GP1:91,2] = PR[GP1:90,2] + 38.049;
   1:L PR[91] 10mm/sec CNT100;
   1:  PR[GP1:91,1] = PR[GP1:90,1] + -34.601;
   1:  PR[GP1:91,2] = PR[GP1:90,2] + 36.973;
   1:L PR[91] 10mm/sec CNT100;
   1:  PR[GP1:91,1] = PR[GP1:90,1] + -42.455;
   1:  PR[GP1:91,2] = PR[GP1:90,2] + 33.538;
   1:L PR[91] 10mm/sec CNT100;
   1:  PR[GP1:91,1] = PR[GP1:90,1] + -45.315;
   1:  PR[GP1:91,2] = PR[GP1:90,2] + 31.735;
   1:L PR[91] 10mm/sec CNT100;
   1:  PR[GP1:91,1] = PR[GP1:90,1] + -47.925;
   1:  PR[GP1:91,2] = PR[GP1:90,2] + 29.187;
   1:L PR[91] 10mm/sec CNT100;
   1:  PR[GP1:91,1] = PR[GP1:90,1] + -53.661;
   1:  PR[GP1:91,2] = PR[GP1:90,2] + 23.994;
   1:L PR[91] 10mm/sec CNT100;
   1:  PR[GP1:91,1] = PR[GP1:90,1] + -55.731;
   1:  PR[GP1:91,2] = PR[GP1:90,2] + 20.764;
   1:L PR[91] 10mm/sec CNT100;
   1:  PR[GP1:91,1] = PR[GP1:90,1] + -59.197;
   1:  PR[GP1:91,2] = PR[GP1:90,2] + 14.502;
   1:L PR[91] 10mm/sec CNT100;
   1:  PR[GP1:91,1] = PR[GP1:90,1] + -60.526;
   1:  PR[GP1:91,2] = PR[GP1:90,2] + 10.840;
   1:L PR[91] 10mm/sec CNT100;
   1:  PR[GP1:91,1] = PR[GP1:90,1] + -60.958;
   1:  PR[GP1:91,2] = PR[GP1:90,2] + 6.983;
   1:L PR[91] 10mm/sec CNT100;
   1:  PR[GP1:91,1] = PR[GP1:90,1] + -62.109;
   1:  PR[GP1:91,2] = PR[GP1:90,2] + 0.261;
   1:L PR[91] 10mm/sec CNT100;
   1:  PR[GP1:91,1] = PR[GP1:90,1] + -61.685;
   1:  PR[GP1:91,2] = PR[GP1:90,2] + -3.543;
   1:L PR[91] 10mm/sec CNT100;
   1:  PR[GP1:91,1] = PR[GP1:90,1] + -60.537;
   1:  PR[GP1:91,2] = PR[GP1:90,2] + -10.252;
   1:L PR[91] 10mm/sec CNT100;
   1:  PR[GP1:91,1] = PR[GP1:90,1] + -59.202;
   1:  PR[GP1:91,2] = PR[GP1:90,2] + -13.930;
   1:L PR[91] 10mm/sec CNT100;
   1:  PR[GP1:91,1] = PR[GP1:90,1] + -55.751;
   1:  PR[GP1:91,2] = PR[GP1:90,2] + -20.180;
   1:L PR[91] 10mm/sec CNT100;
   1:  PR[GP1:91,1] = PR[GP1:90,1] + -53.675;
   1:  PR[GP1:91,2] = PR[GP1:90,2] + -23.420;
   1:L PR[91] 10mm/sec CNT100;
   1:  PR[GP1:91,1] = PR[GP1:90,1] + -51.147;
   1:  PR[GP1:91,2] = PR[GP1:90,2] + -25.901;
   1:L PR[91] 10mm/sec CNT100;
   1:  PR[GP1:91,1] = PR[GP1:90,1] + -45.369;
   1:  PR[GP1:91,2] = PR[GP1:90,2] + -31.142;
   1:L PR[91] 10mm/sec CNT100;
   1:  PR[GP1:91,1] = PR[GP1:90,1] + -42.500;
   1:  PR[GP1:91,2] = PR[GP1:90,2] + -32.951;
   1:L PR[91] 10mm/sec CNT100;
   1:  PR[GP1:91,1] = PR[GP1:90,1] + -34.675;
   1:  PR[GP1:91,2] = PR[GP1:90,2] + -36.395;
   1:L PR[91] 10mm/sec CNT100;
   1:  PR[GP1:91,1] = PR[GP1:90,1] + -31.724;
   1:  PR[GP1:91,2] = PR[GP1:90,2] + -37.476;
   1:L PR[91] 10mm/sec CNT100;
   1:  PR[GP1:91,1] = PR[GP1:90,1] + -28.918;
   1:  PR[GP1:91,2] = PR[GP1:90,2] + -37.875;
   1:L PR[91] 10mm/sec CNT100;
   1:  PR[GP1:91,1] = PR[GP1:90,1] + -19.599;
   1:  PR[GP1:91,2] = PR[GP1:90,2] + -38.769;
   1:L PR[91] 10mm/sec CNT100;
   1:  PR[GP1:91,1] = PR[GP1:90,1] + -17.090;
   1:  PR[GP1:91,2] = PR[GP1:90,2] + -38.604;
   1:L PR[91] 10mm/sec CNT100;
   1:  PR[GP1:91,1] = PR[GP1:90,1] + -7.267;
   1:  PR[GP1:91,2] = PR[GP1:90,2] + -36.356;
   1:L PR[91] 10mm/sec CNT100;
   1:  PR[GP1:91,1] = PR[GP1:90,1] + -5.153;
   1:  PR[GP1:91,2] = PR[GP1:90,2] + -35.749;
   1:L PR[91] 10mm/sec CNT100;
   1:  PR[GP1:91,1] = PR[GP1:90,1] + -0.266;
   1:  PR[GP1:91,2] = PR[GP1:90,2] + -32.886;
   1:L PR[91] 10mm/sec CNT100;
   1:  PR[GP1:91,1] = PR[GP1:90,1] + 4.370;
   1:  PR[GP1:91,2] = PR[GP1:90,2] + -35.818;
   1:  PR[GP1:91,3] = PR[GP1:90,3] + 74.115;
   1:L PR[91] 10mm/sec CNT100;
   1:  PR[GP1:91,1] = PR[GP1:90,1] + 6.366;
   1:  PR[GP1:91,2] = PR[GP1:90,2] + -36.391;
   1:L PR[91] 10mm/sec CNT100;
   1:  PR[GP1:91,1] = PR[GP1:90,1] + 16.388;
   1:  PR[GP1:91,2] = PR[GP1:90,2] + -38.684;
   1:L PR[91] 10mm/sec CNT100;
   1:  PR[GP1:91,1] = PR[GP1:90,1] + 18.754;
   1:  PR[GP1:91,2] = PR[GP1:90,2] + -38.841;
   1:L PR[91] 10mm/sec CNT100;
   1:  PR[GP1:91,1] = PR[GP1:90,1] + 21.441;
   1:  PR[GP1:91,2] = PR[GP1:90,2] + -38.470;
   1:L PR[91] 10mm/sec CNT100;
   1:  PR[GP1:91,1] = PR[GP1:90,1] + 30.977;
   1:  PR[GP1:91,2] = PR[GP1:90,2] + -37.544;
   1:L PR[91] 10mm/sec CNT100;
   1:  PR[GP1:91,1] = PR[GP1:90,1] + 33.793;
   1:  PR[GP1:91,2] = PR[GP1:90,2] + -36.516;
   1:L PR[91] 10mm/sec CNT100;
   1:  PR[GP1:91,1] = PR[GP1:90,1] + 41.817;
   1:  PR[GP1:91,2] = PR[GP1:90,2] + -32.987;
   1:L PR[91] 10mm/sec CNT100;
   1:  PR[GP1:91,1] = PR[GP1:90,1] + 44.549;
   1:  PR[GP1:91,2] = PR[GP1:90,2] + -31.273;
   1:L PR[91] 10mm/sec CNT100;
   1:  PR[GP1:91,1] = PR[GP1:90,1] + 47.054;
   1:  PR[GP1:91,2] = PR[GP1:90,2] + -28.832;
   1:L PR[91] 10mm/sec CNT100;
   1:  PR[GP1:91,1] = PR[GP1:90,1] + 52.935;
   1:  PR[GP1:91,2] = PR[GP1:90,2] + -23.482;
   1:L PR[91] 10mm/sec CNT100;
   1:  PR[GP1:91,1] = PR[GP1:90,1] + 54.952;
   1:  PR[GP1:91,2] = PR[GP1:90,2] + -20.353;
   1:L PR[91] 10mm/sec CNT100;
   1:  PR[GP1:91,1] = PR[GP1:90,1] + 58.512;
   1:  PR[GP1:91,2] = PR[GP1:90,2] + -13.919;
   1:L PR[91] 10mm/sec CNT100;
   1:  PR[GP1:91,1] = PR[GP1:90,1] + 59.790;
   1:  PR[GP1:91,2] = PR[GP1:90,2] + -10.445;
   1:L PR[91] 10mm/sec CNT100;
   1:  PR[GP1:91,1] = PR[GP1:90,1] + 60.222;
   1:  PR[GP1:91,2] = PR[GP1:90,2] + -6.637;
   1:L PR[91] 10mm/sec CNT100;
   1:  PR[GP1:91,1] = PR[GP1:90,1] + 61.405;
   1:  PR[GP1:91,2] = PR[GP1:90,2] + 0.296;
   1:L PR[91] 10mm/sec CNT100;
   1:  PR[GP1:91,1] = PR[GP1:90,1] + 60.980;
   1:  PR[GP1:91,2] = PR[GP1:90,2] + 4.053;
   1:L PR[91] 10mm/sec CNT100;
   1:  PR[GP1:91,1] = PR[GP1:90,1] + 59.790;
   1:  PR[GP1:91,2] = PR[GP1:90,2] + 11.001;
   1:L PR[91] 10mm/sec CNT100;
   1:  PR[GP1:91,1] = PR[GP1:90,1] + 58.507;
   1:  PR[GP1:91,2] = PR[GP1:90,2] + 14.492;
   1:L PR[91] 10mm/sec CNT100;
   1:  PR[GP1:91,1] = PR[GP1:90,1] + 54.932;
   1:  PR[GP1:91,2] = PR[GP1:90,2] + 20.937;
   1:L PR[91] 10mm/sec CNT100;
   1:  PR[GP1:91,1] = PR[GP1:90,1] + 52.908;
   1:  PR[GP1:91,2] = PR[GP1:90,2] + 24.075;
   1:L PR[91] 10mm/sec CNT100;
   1:  PR[GP1:91,1] = PR[GP1:90,1] + 50.474;
   1:  PR[GP1:91,2] = PR[GP1:90,2] + 26.459;
   1:L PR[91] 10mm/sec CNT100;
   1:  PR[GP1:91,1] = PR[GP1:90,1] + 44.513;
   1:  PR[GP1:91,2] = PR[GP1:90,2] + 31.855;
   1:L PR[91] 10mm/sec CNT100;
   1:  PR[GP1:91,1] = PR[GP1:90,1] + 41.771;
   1:  PR[GP1:91,2] = PR[GP1:90,2] + 33.575;
   1:L PR[91] 10mm/sec CNT100;
   1:  PR[GP1:91,1] = PR[GP1:90,1] + 33.717;
   1:  PR[GP1:91,2] = PR[GP1:90,2] + 37.094;
   1:L PR[91] 10mm/sec CNT100;
   1:  PR[GP1:91,1] = PR[GP1:90,1] + 30.887;
   1:  PR[GP1:91,2] = PR[GP1:90,2] + 38.126;
   1:L PR[91] 10mm/sec CNT100;
   1:  PR[GP1:91,1] = PR[GP1:90,1] + 28.211;
   1:  PR[GP1:91,2] = PR[GP1:90,2] + 38.506;
   1:L PR[91] 10mm/sec CNT100;
   1:  PR[GP1:91,1] = PR[GP1:90,1] + 18.659;
   1:  PR[GP1:91,2] = PR[GP1:90,2] + 39.393;
   1:L PR[91] 10mm/sec CNT100;
   1:  PR[GP1:91,1] = PR[GP1:90,1] + 16.283;
   1:  PR[GP1:91,2] = PR[GP1:90,2] + 39.236;
   1:L PR[91] 10mm/sec CNT100;
   1:  PR[GP1:91,1] = PR[GP1:90,1] + 6.096;
   1:  PR[GP1:91,2] = PR[GP1:90,2] + 36.830;
   1:L PR[91] 10mm/sec CNT100;
   1:  PR[GP1:91,1] = PR[GP1:90,1] + 4.172;
   1:  PR[GP1:91,2] = PR[GP1:90,2] + 36.276;
   1:L PR[91] 10mm/sec CNT100;
   1:  PR[GP1:91,1] = PR[GP1:90,1] + 1.746;
   1:  PR[GP1:91,2] = PR[GP1:90,2] + 34.988;
   1:L PR[91] 10mm/sec CNT100;
   1:  PR[GP1:91,1] = PR[GP1:90,1] + -0.263;
   1:  PR[GP1:91,2] = PR[GP1:90,2] + 33.354;
   1:L PR[91] 10mm/sec CNT100;
   1:  PR[GP1:91,1] = PR[GP1:90,1] + -2.268;
   1:  PR[GP1:91,2] = PR[GP1:90,2] + 34.984;
   1:L PR[91] 10mm/sec CNT100;
   1:  PR[GP1:91,1] = PR[GP1:90,1] + -4.696;
   1:  PR[GP1:91,2] = PR[GP1:90,2] + 36.277;
   1:L PR[91] 10mm/sec CNT100;
   1:  PR[GP1:91,1] = PR[GP1:90,1] + -6.618;
   1:  PR[GP1:91,2] = PR[GP1:90,2] + 36.830;
   1:L PR[91] 10mm/sec CNT100;
   1:  PR[GP1:91,1] = PR[GP1:90,1] + -16.808;
   1:  PR[GP1:91,2] = PR[GP1:90,2] + 39.235;
   1:L PR[91] 10mm/sec CNT100;
   1:  PR[GP1:91,1] = PR[GP1:90,1] + -19.178;
   1:  PR[GP1:91,2] = PR[GP1:90,2] + 39.392;
   1:L PR[91] 10mm/sec CNT100;
   1:  PR[GP1:91,1] = PR[GP1:90,1] + -21.874;
   1:  PR[GP1:91,2] = PR[GP1:90,2] + 39.019;
   1:L PR[91] 10mm/sec CNT100;
   1:  PR[GP1:91,1] = PR[GP1:90,1] + -31.442;
   1:  PR[GP1:91,2] = PR[GP1:90,2] + 38.119;
   1:L PR[91] 10mm/sec CNT100;
   1:  PR[GP1:91,1] = PR[GP1:90,1] + -34.254;
   1:  PR[GP1:91,2] = PR[GP1:90,2] + 37.089;
   1:L PR[91] 10mm/sec CNT100;
   1:  PR[GP1:91,1] = PR[GP1:90,1] + -42.309;
   1:  PR[GP1:91,2] = PR[GP1:90,2] + 33.568;
   1:L PR[91] 10mm/sec CNT100;
   1:  PR[GP1:91,1] = PR[GP1:90,1] + -45.057;
   1:  PR[GP1:91,2] = PR[GP1:90,2] + 31.835;
   1:L PR[91] 10mm/sec CNT100;
   1:  PR[GP1:91,1] = PR[GP1:90,1] + -47.568;
   1:  PR[GP1:91,2] = PR[GP1:90,2] + 29.384;
   1:L PR[91] 10mm/sec CNT100;
   1:  PR[GP1:91,1] = PR[GP1:90,1] + -53.473;
   1:  PR[GP1:91,2] = PR[GP1:90,2] + 24.037;
   1:L PR[91] 10mm/sec CNT100;
   1:  PR[GP1:91,1] = PR[GP1:90,1] + -55.468;
   1:  PR[GP1:91,2] = PR[GP1:90,2] + 20.923;
   1:L PR[91] 10mm/sec CNT100;
   1:  PR[GP1:91,1] = PR[GP1:90,1] + -59.043;
   1:  PR[GP1:91,2] = PR[GP1:90,2] + 14.466;
   1:L PR[91] 10mm/sec CNT100;
   1:  PR[GP1:91,1] = PR[GP1:90,1] + -60.326;
   1:  PR[GP1:91,2] = PR[GP1:90,2] + 10.930;
   1:L PR[91] 10mm/sec CNT100;
   1:  PR[GP1:91,1] = PR[GP1:90,1] + -60.743;
   1:  PR[GP1:91,2] = PR[GP1:90,2] + 7.203;
   1:L PR[91] 10mm/sec CNT100;
   1:  PR[GP1:91,1] = PR[GP1:90,1] + -61.931;
   1:  PR[GP1:91,2] = PR[GP1:90,2] + 0.261;
   1:L PR[91] 10mm/sec CNT100;
   1:  PR[GP1:91,1] = PR[GP1:90,1] + -61.522;
   1:  PR[GP1:91,2] = PR[GP1:90,2] + -3.415;
   1:L PR[91] 10mm/sec CNT100;
   1:  PR[GP1:91,1] = PR[GP1:90,1] + -60.337;
   1:  PR[GP1:91,2] = PR[GP1:90,2] + -10.341;
   1:L PR[91] 10mm/sec CNT100;
   1:  PR[GP1:91,1] = PR[GP1:90,1] + -59.048;
   1:  PR[GP1:91,2] = PR[GP1:90,2] + -13.894;
   1:L PR[91] 10mm/sec CNT100;
   1:  PR[GP1:91,1] = PR[GP1:90,1] + -55.489;
   1:  PR[GP1:91,2] = PR[GP1:90,2] + -20.339;
   1:L PR[91] 10mm/sec CNT100;
   1:  PR[GP1:91,1] = PR[GP1:90,1] + -53.487;
   1:  PR[GP1:91,2] = PR[GP1:90,2] + -23.463;
   1:L PR[91] 10mm/sec CNT100;
   1:  PR[GP1:91,1] = PR[GP1:90,1] + -51.049;
   1:  PR[GP1:91,2] = PR[GP1:90,2] + -25.855;
   1:L PR[91] 10mm/sec CNT100;
   1:  PR[GP1:91,1] = PR[GP1:90,1] + -45.112;
   1:  PR[GP1:91,2] = PR[GP1:90,2] + -31.241;
   1:L PR[91] 10mm/sec CNT100;
   1:  PR[GP1:91,1] = PR[GP1:90,1] + -42.354;
   1:  PR[GP1:91,2] = PR[GP1:90,2] + -32.980;
   1:L PR[91] 10mm/sec CNT100;
   1:  PR[GP1:91,1] = PR[GP1:90,1] + -34.331;
   1:  PR[GP1:91,2] = PR[GP1:90,2] + -36.511;
   1:L PR[91] 10mm/sec CNT100;
   1:  PR[GP1:91,1] = PR[GP1:90,1] + -31.506;
   1:  PR[GP1:91,2] = PR[GP1:90,2] + -37.546;
   1:L PR[91] 10mm/sec CNT100;
   1:  PR[GP1:91,1] = PR[GP1:90,1] + -28.820;
   1:  PR[GP1:91,2] = PR[GP1:90,2] + -37.928;
   1:L PR[91] 10mm/sec CNT100;
   1:  PR[GP1:91,1] = PR[GP1:90,1] + -19.299;
   1:  PR[GP1:91,2] = PR[GP1:90,2] + -38.841;
   1:L PR[91] 10mm/sec CNT100;
   1:  PR[GP1:91,1] = PR[GP1:90,1] + -16.914;
   1:  PR[GP1:91,2] = PR[GP1:90,2] + -38.684;
   1:L PR[91] 10mm/sec CNT100;
   1:  PR[GP1:91,1] = PR[GP1:90,1] + -6.891;
   1:  PR[GP1:91,2] = PR[GP1:90,2] + -36.391;
   1:L PR[91] 10mm/sec CNT100;
   1:  PR[GP1:91,1] = PR[GP1:90,1] + -4.898;
   1:  PR[GP1:91,2] = PR[GP1:90,2] + -35.819;
   1:L PR[91] 10mm/sec CNT100;
   1:  PR[GP1:91,1] = PR[GP1:90,1] + -0.266;
   1:  PR[GP1:91,2] = PR[GP1:90,2] + -33.105;
   1:L PR[91] 10mm/sec CNT100;
   1:  PR[GP1:91,1] = PR[GP1:90,1] + 4.115;
   1:  PR[GP1:91,2] = PR[GP1:90,2] + -35.887;
   1:  PR[GP1:91,3] = PR[GP1:90,3] + 74.725;
   1:L PR[91] 10mm/sec CNT100;
   1:  PR[GP1:91,1] = PR[GP1:90,1] + 5.990;
   1:  PR[GP1:91,2] = PR[GP1:90,2] + -36.426;
   1:L PR[91] 10mm/sec CNT100;
   1:  PR[GP1:91,1] = PR[GP1:90,1] + 16.211;
   1:  PR[GP1:91,2] = PR[GP1:90,2] + -38.764;
   1:L PR[91] 10mm/sec CNT100;
   1:  PR[GP1:91,1] = PR[GP1:90,1] + 18.454;
   1:  PR[GP1:91,2] = PR[GP1:90,2] + -38.913;
   1:L PR[91] 10mm/sec CNT100;
   1:  PR[GP1:91,1] = PR[GP1:90,1] + 21.005;
   1:  PR[GP1:91,2] = PR[GP1:90,2] + -38.561;
   1:L PR[91] 10mm/sec CNT100;
   1:  PR[GP1:91,1] = PR[GP1:90,1] + 30.759;
   1:  PR[GP1:91,2] = PR[GP1:90,2] + -37.613;
   1:L PR[91] 10mm/sec CNT100;
